KUKA KRL program: EPS_2_25252_SD2A_A_20250910061719.src

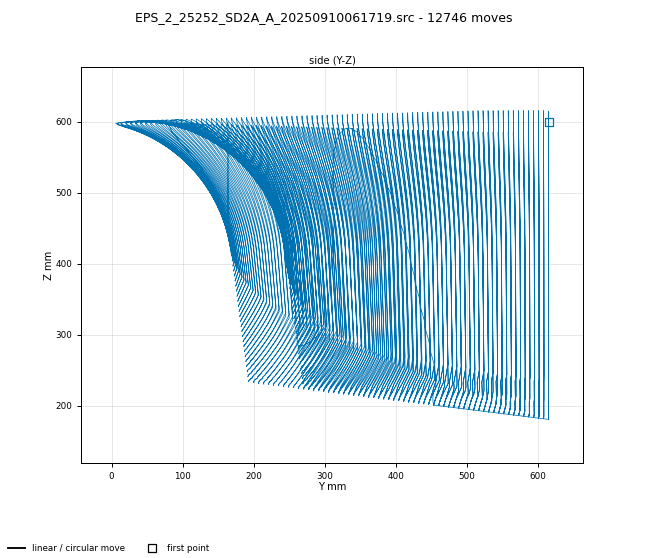
[picture p0: tool path of EPS_2_25252_SD2A_A_20250910061719.src, 12746 of 12748 moves have a stored position in this frame; points joined in program order, loops and branches not executed]
&ACCESS RVP
&REL 4
&COMMENT QRS 19112012
&PARAM EDITMASK = *
DEF PART()
EXT BAS (BAS_COMMAND :IN,REAL :IN )
INT I
BAS (#INITMOV,0 )

;KUKA QRS Post kuka4.cps  Date:22-06-2017 !

File_ID=2823

QRS_PRE_INIT()

;Init var - Until changes are made in qrs_pre_init
Outlet_Square_prg=0
Inlet_1_Square_prg=0
Inlet_2_Square_prg=0
Inlet_3_Square_prg=0
Inlet_4_Square_prg=0
Inlet_5_Square_prg=0

Outlet_1={X 0.000, Y 518.380, Z 433.000, B 0.000, E1 0.000 }
Inlet_1={X 0.000, Y 520.620, Z 403.000, B 0.000, E1 206.000 }
Outlet_1_type=366
Inlet_1_type=366
;QRS#1=Sidecore dimensions
;QRS#2=375-15" PVC SDR 35
;QRS#3=375-15" PVC SDR 35
;QRS#4=
;QRS#5=
;QRS#6=
;QRS#7=
;QRS#8=
;QRS#9=20Y PSX
;QRS#10=20Y PSX
;QRS#11=
;QRS#12=
;QRS#13=
;QRS#14=
;QRS#15=
;QRS#16=1220x127x914 3'
;QRS#17=EPS Height
;QRS#18=616
;QRS#19=*
;QRS#20= UPDATED VERSION 22-06-2017
;QRS#21=*
Outlet_Square=0250
Inlet_1_Square=0250
Inlet_2_Square=0
Inlet_3_Square=0
Inlet_4_Square=0
Inlet_5_Square=0
Mill_Square=1
Outlet_Square_Prg=252
Inlet_1_Square_prg=252

QRS_INIT()

$ADVANCE=5

; T1
PTP {E1 173.604,E2 173.604}
PTP {X 0,Y 615.505,A -85,B 0,C 180,E1 173.604,E2 173.604,E3 0,E4 0,E5 0,E6 0}
QRS_SPEED_INIT()
LIN {X 0,Y 615.505,Z 600,A -85,B 0,C 180,E1 173.604,E2 173.604,E3 0,E4 0,E5 0,E6 0} C_VEL
LIN {X 0,Y 615.505,Z 191.184,A -85,B 0,C 180,E1 173.604,E2 173.604} C_VEL
LIN {X 0,Y 615.505,Z 183.002,A -85,B 0,C 180,E1 173.604,E2 173.604} C_VEL
LIN {X 0,Y 615.487,Z 181.002,A -85,B 0,C 180,E1 173.418,E2 173.418} C_VEL
LIN {X 0,Y 615.475,Z 180.998,A -85,B 0,C 180,E1 170.801,E2 170.801} C_VEL
LIN {X 0,Y 615.481,Z 181.009,A -85,B 0,C 180,E1 168.139,E2 168.139} C_VEL
LIN {X 0,Y 615.486,Z 181,A -85,B 0,C 180,E1 165.451,E2 165.451} C_VEL
LIN {X 0,Y 615.47,Z 181.001,A -85,B 0,C 180,E1 162.729,E2 162.729} C_VEL
LIN {X 0,Y 615.488,Z 181.012,A -85,B 0,C 180,E1 159.967,E2 159.967} C_VEL
LIN {X 0,Y 615.49,Z 180.994,A -85,B 0,C 180,E1 157.156,E2 157.156} C_VEL
LIN {X 0,Y 615.489,Z 181.01,A -85,B 0,C 180,E1 154.284,E2 154.284} C_VEL
LIN {X 0,Y 615.487,Z 180.995,A -85,B 0,C 180,E1 151.342,E2 151.342} C_VEL
LIN {X 0,Y 615.474,Z 181,A -85,B 0,C 180,E1 148.915,E2 148.915} C_VEL
LIN {X 0,Y 615.485,Z 181.009,A -85,B 0,C 180,E1 146.465,E2 146.465} C_VEL
LIN {X 0,Y 615.482,Z 180.997,A -85,B 0,C 180,E1 143.575,E2 143.575} C_VEL
LIN {X 0,Y 615.474,Z 181.002,A -85,B 0,C 180,E1 140.939,E2 140.939} C_VEL
LIN {X 0,Y 615.488,Z 181.011,A -85,B 0,C 180,E1 138.526,E2 138.526} C_VEL
LIN {X 0,Y 615.477,Z 181,A -85,B 0,C 180,E1 135.85,E2 135.85} C_VEL
LIN {X 0,Y 615.477,Z 181.002,A -85,B 0,C 180,E1 133.047,E2 133.047} C_VEL
LIN {X 0,Y 615.491,Z 181.013,A -85,B 0,C 180,E1 130.606,E2 130.606} C_VEL
LIN {X 0,Y 615.477,Z 181.001,A -85,B 0,C 180,E1 128.011,E2 128.011} C_VEL
LIN {X 0,Y 615.497,Z 180.993,A -85,B 0,C 180,E1 125.615,E2 125.615} C_VEL
LIN {X 0,Y 615.48,Z 181.001,A -85,B 0,C 180,E1 123.236,E2 123.236} C_VEL
LIN {X 0,Y 615.486,Z 181.008,A -85,B 0,C 180,E1 120.92,E2 120.92} C_VEL
LIN {X 0,Y 615.476,Z 181.007,A -85,B 0,C 180,E1 118.449,E2 118.449} C_VEL
LIN {X 0,Y 615.489,Z 180.996,A -85,B 0,C 180,E1 115.569,E2 115.569} C_VEL
LIN {X 0,Y 615.487,Z 181.015,A -85,B 0,C 180,E1 112.844,E2 112.844} C_VEL
LIN {X 0,Y 615.48,Z 180.997,A -85,B 0,C 180,E1 110.033,E2 110.033} C_VEL
LIN {X 0,Y 615.484,Z 181.005,A -85,B 0,C 180,E1 107.271,E2 107.271} C_VEL
LIN {X 0,Y 615.472,Z 181.005,A -85,B 0,C 180,E1 104.549,E2 104.549} C_VEL
LIN {X 0,Y 615.486,Z 180.996,A -85,B 0,C 180,E1 101.861,E2 101.861} C_VEL
LIN {X 0,Y 615.489,Z 181.01,A -85,B 0,C 180,E1 99.199,E2 99.199} C_VEL
LIN {X 0,Y 615.468,Z 181.003,A -85,B 0,C 180,E1 96.557,E2 96.557} C_VEL
LIN {X 0,Y 615.487,Z 180.996,A -85,B 0,C 180,E1 93.929,E2 93.929} C_VEL
LIN {X 0,Y 615.489,Z 181.011,A -85,B 0,C 180,E1 91.309,E2 91.309} C_VEL
LIN {X 0,Y 615.465,Z 181.004,A -85,B 0,C 180,E1 88.692,E2 88.692} C_VEL
LIN {X 0,Y 615.48,Z 181.04,A -85,B 0,C 180,E1 88.242,E2 88.242} C_VEL
LIN {X 0,Y 615.493,Z 205.876,A -85,B 0,C 180,E1 85.969,E2 85.969} C_VEL
LIN {X 0,Y 615.49,Z 411.015,A -85,B 0,C 180,E1 83.444,E2 83.444} C_VEL
LIN {X 0,Y 615.494,Z 426.259,A -85,B 0,C 180,E1 83.141,E2 83.141} C_VEL
LIN {X 0,Y 615.491,Z 442.192,A -85,B 0,C 180,E1 82.702,E2 82.702} C_VEL
LIN {X 0,Y 615.493,Z 458.161,A -85,B 0,C 180,E1 82.125,E2 82.125} C_VEL
LIN {X 0,Y 615.492,Z 472.639,A -85,B 0,C 180,E1 81.464,E2 81.464} C_VEL
LIN {X 0,Y 615.498,Z 487.682,A -85,B 0,C 180,E1 80.636,E2 80.636} C_VEL
LIN {X 0,Y 615.495,Z 501.587,A -85,B 0,C 180,E1 79.723,E2 79.723} C_VEL
LIN {X 0,Y 615.496,Z 513.498,A -85,B 0,C 180,E1 78.807,E2 78.807} C_VEL
LIN {X 0,Y 615.493,Z 526.453,A -85,B 0,C 180,E1 77.638,E2 77.638} C_VEL
LIN {X 0,Y 615.498,Z 537.483,A -85,B 0,C 180,E1 76.463,E2 76.463} C_VEL
LIN {X 0,Y 615.491,Z 547.006,A -85,B 0,C 180,E1 75.282,E2 75.282} C_VEL
LIN {X 0,Y 615.492,Z 555.274,A -85,B 0,C 180,E1 74.095,E2 74.095} C_VEL
LIN {X 0,Y 615.49,Z 563.212,A -85,B 0,C 180,E1 72.73,E2 72.73} C_VEL
LIN {X 0,Y 615.491,Z 569.836,A -85,B 0,C 180,E1 71.355,E2 71.355} C_VEL
LIN {X 0,Y 615.491,Z 575.27,A -85,B 0,C 180,E1 69.968,E2 69.968} C_VEL
LIN {X 0,Y 615.497,Z 579.442,A -85,B 0,C 180,E1 68.569,E2 68.569} C_VEL
LIN {X 0,Y 615.485,Z 582.529,A -85,B 0,C 180,E1 67.156,E2 67.156} C_VEL
LIN {X 0,Y 615.486,Z 584.519,A -85,B 0,C 180,E1 65.728,E2 65.728} C_VEL
LIN {X 0,Y 615.5,Z 585.313,A -85,B 0,C 180,E1 64.285,E2 64.285} C_VEL
LIN {X 0,Y 615.485,Z 584.997,A -85,B 0,C 180,E1 62.823,E2 62.823} C_VEL
LIN {X 0,Y 615.485,Z 583.512,A -85,B 0,C 180,E1 61.343,E2 61.343} C_VEL
LIN {X 0,Y 615.486,Z 580.675,A -85,B 0,C 180,E1 59.84,E2 59.84} C_VEL
LIN {X 0,Y 615.495,Z 576.462,A -85,B 0,C 180,E1 58.316,E2 58.316} C_VEL
LIN {X 0,Y 615.488,Z 570.734,A -85,B 0,C 180,E1 56.765,E2 56.765} C_VEL
LIN {X 0,Y 615.49,Z 565.578,A -85,B 0,C 180,E1 55.64,E2 55.64} C_VEL
LIN {X 0,Y 615.499,Z 558.745,A -85,B 0,C 180,E1 54.386,E2 54.386} C_VEL
LIN {X 0,Y 615.492,Z 550.22,A -85,B 0,C 180,E1 53.063,E2 53.063} C_VEL
LIN {X 0,Y 615.494,Z 539.889,A -85,B 0,C 180,E1 51.725,E2 51.725} C_VEL
LIN {X 0,Y 615.499,Z 527.977,A -85,B 0,C 180,E1 50.424,E2 50.424} C_VEL
LIN {X 0,Y 615.493,Z 515.499,A -85,B 0,C 180,E1 49.273,E2 49.273} C_VEL
LIN {X 0,Y 615.499,Z 503.131,A -85,B 0,C 180,E1 48.3,E2 48.3} C_VEL
LIN {X 0,Y 615.495,Z 489.57,A -85,B 0,C 180,E1 47.388,E2 47.388} C_VEL
LIN {X 0,Y 615.493,Z 475.141,A -85,B 0,C 180,E1 46.569,E2 46.569} C_VEL
LIN {X 0,Y 615.493,Z 459.721,A -85,B 0,C 180,E1 45.852,E2 45.852} C_VEL
LIN {X 0,Y 615.496,Z 445.386,A -85,B 0,C 180,E1 45.315,E2 45.315} C_VEL
LIN {X 0,Y 615.49,Z 429.017,A -85,B 0,C 180,E1 44.834,E2 44.834} C_VEL
LIN {X 0,Y 615.494,Z 412.614,A -85,B 0,C 180,E1 44.49,E2 44.49} C_VEL
LIN {X 0,Y 615.451,Z 290.429,A -85,B 0,C 180,E1 42.979,E2 42.979} C_VEL
LIN {X 0,Y 615.445,Z 205.76,A -85,B 0,C 180,E1 41.928,E2 41.928} C_VEL
LIN {X 0,Y 615.419,Z 181.064,A -85,B 0,C 180,E1 39.668,E2 39.668} C_VEL
LIN {X 0,Y 615.463,Z 181.013,A -85,B 0,C 180,E1 36.935,E2 36.935} C_VEL
LIN {X 0,Y 615.496,Z 181.01,A -85,B 0,C 180,E1 34.703,E2 34.703} C_VEL
LIN {X 0,Y 615.426,Z 181.01,A -85,B 0,C 180,E1 31.689,E2 31.689} C_VEL
LIN {X 0,Y 615.444,Z 181.01,A -85,B 0,C 180,E1 29.408,E2 29.408} C_VEL
LIN {X 0,Y 615.462,Z 181.005,A -85,B 0,C 180,E1 26.445,E2 26.445} C_VEL
LIN {X 0,Y 615.437,Z 181.007,A -85,B 0,C 180,E1 24,E2 24} C_VEL
LIN {X 0,Y 615.442,Z 181.006,A -85,B 0,C 180,E1 22.138,E2 22.138} C_VEL
LIN {X 0,Y 615.439,Z 181.007,A -85,B 0,C 180,E1 20.034,E2 20.034} C_VEL
LIN {X 0,Y 615.491,Z 181.013,A -85,B 0,C 180,E1 17.27,E2 17.27} C_VEL
LIN {X 0,Y 615.468,Z 181.001,A -85,B 0,C 180,E1 14.549,E2 14.549} C_VEL
LIN {X 0,Y 615.465,Z 181.001,A -85,B 0,C 180,E1 12.531,E2 12.531} C_VEL
LIN {X 0,Y 615.46,Z 181.008,A -85,B 0,C 180,E1 9.863,E2 9.863} C_VEL
LIN {X 0,Y 615.493,Z 181.005,A -85,B 0,C 180,E1 7.216,E2 7.216} C_VEL
LIN {X 0,Y 615.462,Z 181.001,A -85,B 0,C 180,E1 4.585,E2 4.585} C_VEL
LIN {X 0,Y 615.47,Z 181.008,A -85,B 0,C 180,E1 1.963,E2 1.963} C_VEL
LIN {X 0,Y 615.489,Z 181.003,A -85,B 0,C 180,E1 -0.654,E2 -0.654} C_VEL
LIN {X 0,Y 615.474,Z 180.999,A -85,B 0,C 180,E1 -3.273,E2 -3.273} C_VEL
LIN {X 0,Y 615.472,Z 181.01,A -85,B 0,C 180,E1 -5.899,E2 -5.899} C_VEL
LIN {X 0,Y 615.484,Z 181.002,A -85,B 0,C 180,E1 -8.537,E2 -8.537} C_VEL
LIN {X 0,Y 615.476,Z 180.998,A -85,B 0,C 180,E1 -11.193,E2 -11.193} C_VEL
LIN {X 0,Y 615.499,Z 181.012,A -85,B 0,C 180,E1 -13.941,E2 -13.941} C_VEL
LIN {X 0,Y 615.486,Z 180.998,A -85,B 0,C 180,E1 -16.587,E2 -16.587} C_VEL
LIN {X 0,Y 615.474,Z 181.004,A -85,B 0,C 180,E1 -19.338,E2 -19.338} C_VEL
LIN {X 0,Y 615.478,Z 181.005,A -85,B 0,C 180,E1 -22.137,E2 -22.137} C_VEL
LIN {X 0,Y 615.483,Z 180.998,A -85,B 0,C 180,E1 -24.992,E2 -24.992} C_VEL
LIN {X 0,Y 615.475,Z 181.007,A -85,B 0,C 180,E1 -27.916,E2 -27.916} C_VEL
LIN {X 0,Y 615.47,Z 181.002,A -85,B 0,C 180,E1 -30.161,E2 -30.161} C_VEL
LIN {X 0,Y 615.484,Z 180.996,A -85,B 0,C 180,E1 -32.458,E2 -32.458} C_VEL
LIN {X 0,Y 615.487,Z 180.999,A -85,B 0,C 180,E1 -34.815,E2 -34.815} C_VEL
LIN {X 0,Y 615.487,Z 181.011,A -85,B 0,C 180,E1 -37.242,E2 -37.242} C_VEL
LIN {X 0,Y 615.466,Z 181.001,A -85,B 0,C 180,E1 -40.088,E2 -40.088} C_VEL
LIN {X 0,Y 615.482,Z 180.997,A -85,B 0,C 180,E1 -42.353,E2 -42.353} C_VEL
LIN {X 0,Y 615.492,Z 181.011,A -85,B 0,C 180,E1 -45.068,E2 -45.068} C_VEL
LIN {X 0,Y 615.458,Z 181.006,A -85,B 0,C 180,E1 -47.645,E2 -47.645} C_VEL
LIN {X 0,Y 615.479,Z 180.998,A -85,B 0,C 180,E1 -50.25,E2 -50.25} C_VEL
LIN {X 0,Y 615.486,Z 181.011,A -85,B 0,C 180,E1 -53.063,E2 -53.063} C_VEL
LIN {X 0,Y 615.458,Z 181.009,A -85,B 0,C 180,E1 -55.303,E2 -55.303} C_VEL
LIN {X 0,Y 615.448,Z 181.005,A -85,B 0,C 180,E1 -57.675,E2 -57.675} C_VEL
LIN {X 0,Y 615.482,Z 181.001,A -85,B 0,C 180,E1 -60.206,E2 -60.206} C_VEL
LIN {X 0,Y 615.468,Z 181.011,A -85,B 0,C 180,E1 -62.958,E2 -62.958} C_VEL
LIN {X 0,Y 615.442,Z 181.191,A -85,B 0,C 180,E1 -63.6,E2 -63.6} C_VEL
LIN {X 0,Y 615.497,Z 213.169,A -85,B 0,C 180,E1 -66.218,E2 -66.218} C_VEL
LIN {X 0,Y 615.485,Z 235.018,A -85,B 0,C 180,E1 -67.974,E2 -67.974} C_VEL
LIN {X 0,Y 615.49,Z 442.459,A -85,B 0,C 180,E1 -70.533,E2 -70.533} C_VEL
LIN {X 0,Y 615.493,Z 459.015,A -85,B 0,C 180,E1 -70.879,E2 -70.879} C_VEL
LIN {X 0,Y 615.492,Z 473.946,A -85,B 0,C 180,E1 -71.311,E2 -71.311} C_VEL
LIN {X 0,Y 615.491,Z 489.356,A -85,B 0,C 180,E1 -71.881,E2 -71.881} C_VEL
LIN {X 0,Y 615.493,Z 504.014,A -85,B 0,C 180,E1 -72.559,E2 -72.559} C_VEL
LIN {X 0,Y 615.5,Z 517.843,A -85,B 0,C 180,E1 -73.329,E2 -73.329} C_VEL
LIN {X 0,Y 615.499,Z 532.043,A -85,B 0,C 180,E1 -74.266,E2 -74.266} C_VEL
LIN {X 0,Y 615.495,Z 545.097,A -85,B 0,C 180,E1 -75.282,E2 -75.282} C_VEL
LIN {X 0,Y 615.494,Z 556.218,A -85,B 0,C 180,E1 -76.295,E2 -76.295} C_VEL
LIN {X 0,Y 615.493,Z 567.294,A -85,B 0,C 180,E1 -77.47,E2 -77.47} C_VEL
LIN {X 0,Y 615.494,Z 576.769,A -85,B 0,C 180,E1 -78.641,E2 -78.641} C_VEL
LIN {X 0,Y 615.496,Z 585.966,A -85,B 0,C 180,E1 -79.972,E2 -79.972} C_VEL
LIN {X 0,Y 615.489,Z 594.503,A -85,B 0,C 180,E1 -81.464,E2 -81.464} C_VEL
LIN {X 0,Y 615.491,Z 601.983,A -85,B 0,C 180,E1 -83.102,E2 -83.102} C_VEL
LIN {X 0,Y 615.492,Z 607.742,A -85,B 0,C 180,E1 -84.759,E2 -84.759} C_VEL
LIN {X 0,Y 615.493,Z 611.077,A -85,B 0,C 180,E1 -86.072,E2 -86.072} C_VEL
LIN {X 0,Y 615.485,Z 613.504,A -85,B 0,C 180,E1 -87.382,E2 -87.382} C_VEL
LIN {X 0,Y 615.488,Z 614.87,A -85,B 0,C 180,E1 -88.692,E2 -88.692} C_VEL
LIN {X 0,Y 615.489,Z 615.39,A -85,B 0,C 180,E1 -90,E2 -90} C_VEL
LIN {X 0,Y 615.488,Z 614.87,A -85,B 0,C 180,E1 -91.309,E2 -91.309} C_VEL
LIN {X 0,Y 615.485,Z 613.504,A -85,B 0,C 180,E1 -92.618,E2 -92.618} C_VEL
LIN {X 0,Y 615.493,Z 611.076,A -85,B 0,C 180,E1 -93.929,E2 -93.929} C_VEL
LIN {X 0,Y 615.492,Z 607.741,A -85,B 0,C 180,E1 -95.241,E2 -95.241} C_VEL
LIN {X 0,Y 615.491,Z 601.982,A -85,B 0,C 180,E1 -96.898,E2 -96.898} C_VEL
LIN {X 0,Y 615.489,Z 594.501,A -85,B 0,C 180,E1 -98.537,E2 -98.537} C_VEL
LIN {X 0,Y 615.496,Z 585.964,A -85,B 0,C 180,E1 -100.028,E2 -100.028} C_VEL
LIN {X 0,Y 615.494,Z 576.766,A -85,B 0,C 180,E1 -101.36,E2 -101.36} C_VEL
LIN {X 0,Y 615.495,Z 567.29,A -85,B 0,C 180,E1 -102.53,E2 -102.53} C_VEL
LIN {X 0,Y 615.496,Z 556.213,A -85,B 0,C 180,E1 -103.706,E2 -103.706} C_VEL
LIN {X 0,Y 615.495,Z 544.115,A -85,B 0,C 180,E1 -104.802,E2 -104.802} C_VEL
LIN {X 0,Y 615.497,Z 529.708,A -85,B 0,C 180,E1 -105.905,E2 -105.905} C_VEL
LIN {X 0,Y 615.497,Z 515.015,A -85,B 0,C 180,E1 -106.842,E2 -106.842} C_VEL
LIN {X 0,Y 615.49,Z 500.511,A -85,B 0,C 180,E1 -107.613,E2 -107.613} C_VEL
LIN {X 0,Y 615.49,Z 485.248,A -85,B 0,C 180,E1 -108.282,E2 -108.282} C_VEL
LIN {X 0,Y 615.49,Z 469.995,A -85,B 0,C 180,E1 -108.819,E2 -108.819} C_VEL
LIN {X 0,Y 615.497,Z 453.521,A -85,B 0,C 180,E1 -109.251,E2 -109.251} C_VEL
LIN {X 0,Y 615.49,Z 437.931,A -85,B 0,C 180,E1 -109.533,E2 -109.533} C_VEL
LIN {X 0,Y 615.485,Z 235.013,A -85,B 0,C 180,E1 -112.026,E2 -112.026} C_VEL
LIN {X 0,Y 615.453,Z 201.612,A -85,B 0,C 180,E1 -114.723,E2 -114.723} C_VEL
LIN {X 0,Y 615.441,Z 181.006,A -85,B 0,C 180,E1 -116.423,E2 -116.423} C_VEL
LIN {X 0,Y 615.443,Z 181.008,A -85,B 0,C 180,E1 -118.66,E2 -118.66} C_VEL
LIN {X 0,Y 615.477,Z 181.011,A -85,B 0,C 180,E1 -121.085,E2 -121.085} C_VEL
LIN {X 0,Y 615.457,Z 181.003,A -85,B 0,C 180,E1 -124.024,E2 -124.024} C_VEL
LIN {X 0,Y 615.444,Z 181.006,A -85,B 0,C 180,E1 -126.427,E2 -126.427} C_VEL
LIN {X 0,Y 615.492,Z 181.012,A -85,B 0,C 180,E1 -129.063,E2 -129.063} C_VEL
LIN {X 0,Y 615.494,Z 181.001,A -85,B 0,C 180,E1 -131.473,E2 -131.473} C_VEL
LIN {X 0,Y 615.448,Z 181.004,A -85,B 0,C 180,E1 -134.153,E2 -134.153} C_VEL
LIN {X 0,Y 615.469,Z 181.011,A -85,B 0,C 180,E1 -136.754,E2 -136.754} C_VEL
LIN {X 0,Y 615.494,Z 181,A -85,B 0,C 180,E1 -139.394,E2 -139.394} C_VEL
LIN {X 0,Y 615.453,Z 181.003,A -85,B 0,C 180,E1 -141.992,E2 -141.992} C_VEL
LIN {X 0,Y 615.454,Z 181.008,A -85,B 0,C 180,E1 -144.382,E2 -144.382} C_VEL
LIN {X 0,Y 615.481,Z 181.014,A -85,B 0,C 180,E1 -146.764,E2 -146.764} C_VEL
LIN {X 0,Y 615.493,Z 181.004,A -85,B 0,C 180,E1 -149.081,E2 -149.081} C_VEL
LIN {X 0,Y 615.474,Z 180.999,A -85,B 0,C 180,E1 -151.551,E2 -151.551} C_VEL
LIN {X 0,Y 615.469,Z 181,A -85,B 0,C 180,E1 -153.555,E2 -153.555} C_VEL
LIN {X 0,Y 615.455,Z 181.004,A -85,B 0,C 180,E1 -155.997,E2 -155.997} C_VEL
LIN {X 0,Y 615.491,Z 181.012,A -85,B 0,C 180,E1 -158.568,E2 -158.568} C_VEL
LIN {X 0,Y 615.477,Z 180.998,A -85,B 0,C 180,E1 -161.396,E2 -161.396} C_VEL
LIN {X 0,Y 615.463,Z 181.007,A -85,B 0,C 180,E1 -164.094,E2 -164.094} C_VEL
LIN {X 0,Y 615.487,Z 181.005,A -85,B 0,C 180,E1 -166.799,E2 -166.799} C_VEL
LIN {X 0,Y 615.468,Z 180.999,A -85,B 0,C 180,E1 -169.473,E2 -169.473} C_VEL
LIN {X 0,Y 615.473,Z 181.009,A -85,B 0,C 180,E1 -172.124,E2 -172.124} C_VEL
LIN {X 0,Y 615.489,Z 181.002,A -85,B 0,C 180,E1 -174.759,E2 -174.759} C_VEL
LIN {X 0,Y 615.47,Z 180.999,A -85,B 0,C 180,E1 -177.382,E2 -177.382} C_VEL
LIN {X 0,Y 615.475,Z 181.009,A -85,B 0,C 180,E1 -180,E2 -180} C_VEL
LIN {X 0,Y 615.488,Z 181.003,A -85,B 0,C 180,E1 -182.618,E2 -182.618} C_VEL
LIN {X 0,Y 615.474,Z 180.998,A -85,B 0,C 180,E1 -185.241,E2 -185.241} C_VEL
LIN {X 0,Y 615.487,Z 181.002,A -85,B 0,C 180,E1 -186.582,E2 -186.582} C_VEL
LIN {X 0,Y 614.803,Z 181.145,A -85,B 0,C 180,E1 -187.128,E2 -187.128} C_VEL
LIN {X 0,Y 611.964,Z 181.571,A -85,B 0,C 180,E1 -188.014,E2 -188.014} C_VEL
LIN {X 0,Y 609.572,Z 181.876,A -85,B 0,C 180,E1 -188.727,E2 -188.727} C_VEL
LIN {X 0,Y 608.538,Z 181.991,A -85,B 0,C 180,E1 -189.276,E2 -189.276} C_VEL
LIN {X 0,Y 608.449,Z 182.002,A -85,B 0,C 180,E1 -189.463,E2 -189.463} C_VEL
LIN {X 0,Y 608.458,Z 182.009,A -85,B 0,C 180,E1 -192,E2 -192} C_VEL
LIN {X 0,Y 608.471,Z 181.999,A -85,B 0,C 180,E1 -194.721,E2 -194.721} C_VEL
LIN {X 0,Y 608.444,Z 182.003,A -85,B 0,C 180,E1 -197.477,E2 -197.477} C_VEL
LIN {X 0,Y 608.463,Z 182.003,A -85,B 0,C 180,E1 -200.274,E2 -200.274} C_VEL
LIN {X 0,Y 608.449,Z 182.001,A -85,B 0,C 180,E1 -203.124,E2 -203.124} C_VEL
LIN {X 0,Y 608.47,Z 182.006,A -85,B 0,C 180,E1 -205.722,E2 -205.722} C_VEL
LIN {X 0,Y 608.473,Z 181.998,A -85,B 0,C 180,E1 -208.621,E2 -208.621} C_VEL
LIN {X 0,Y 608.442,Z 182.005,A -85,B 0,C 180,E1 -211.318,E2 -211.318} C_VEL
LIN {X 0,Y 608.471,Z 182.008,A -85,B 0,C 180,E1 -213.735,E2 -213.735} C_VEL
LIN {X 0,Y 608.474,Z 182.001,A -85,B 0,C 180,E1 -216.09,E2 -216.09} C_VEL
LIN {X 0,Y 608.462,Z 181.998,A -85,B 0,C 180,E1 -218.588,E2 -218.588} C_VEL
LIN {X 0,Y 608.458,Z 182.006,A -85,B 0,C 180,E1 -221.342,E2 -221.342} C_VEL
LIN {X 0,Y 608.447,Z 182.001,A -85,B 0,C 180,E1 -224.263,E2 -224.263} C_VEL
LIN {X 0,Y 608.445,Z 182.004,A -85,B 0,C 180,E1 -227.04,E2 -227.04} C_VEL
LIN {X 0,Y 608.45,Z 182.006,A -85,B 0,C 180,E1 -229.697,E2 -229.697} C_VEL
LIN {X 0,Y 608.462,Z 181.999,A -85,B 0,C 180,E1 -232.254,E2 -232.254} C_VEL
LIN {X 0,Y 608.48,Z 182.002,A -85,B 0,C 180,E1 -235.09,E2 -235.09} C_VEL
LIN {X 0,Y 608.462,Z 182,A -85,B 0,C 180,E1 -237.906,E2 -237.906} C_VEL
LIN {X 0,Y 608.472,Z 181.997,A -85,B 0,C 180,E1 -240.221,E2 -240.221} C_VEL
LIN {X 0,Y 608.476,Z 182.001,A -85,B 0,C 180,E1 -242.793,E2 -242.793} C_VEL
LIN {X 0,Y 608.447,Z 182.007,A -85,B 0,C 180,E1 -245.429,E2 -245.429} C_VEL
LIN {X 0,Y 608.463,Z 181.999,A -85,B 0,C 180,E1 -248.308,E2 -248.308} C_VEL
LIN {X 0,Y 608.466,Z 182.005,A -85,B 0,C 180,E1 -251.285,E2 -251.285} C_VEL
LIN {X 0,Y 608.454,Z 182,A -85,B 0,C 180,E1 -253.906,E2 -253.906} C_VEL
LIN {X 0,Y 608.467,Z 182.002,A -85,B 0,C 180,E1 -256.644,E2 -256.644} C_VEL
LIN {X 0,Y 608.453,Z 182.004,A -85,B 0,C 180,E1 -259.35,E2 -259.35} C_VEL
LIN {X 0,Y 608.476,Z 181.997,A -85,B 0,C 180,E1 -262.033,E2 -262.033} C_VEL
LIN {X 0,Y 608.47,Z 182.006,A -85,B 0,C 180,E1 -264.698,E2 -264.698} C_VEL
LIN {X 0,Y 608.459,Z 182.002,A -85,B 0,C 180,E1 -267.352,E2 -267.352} C_VEL
LIN {X 0,Y 608.477,Z 181.998,A -85,B 0,C 180,E1 -270,E2 -270} C_VEL
LIN {X 0,Y 608.461,Z 182.016,A -85,B 0,C 180,E1 -271.551,E2 -271.551} C_VEL
LIN {X 0,Y 608.729,Z 188.319,A -85,B 0,C 180,E1 -272.15,E2 -272.15} C_VEL
LIN {X 0,Y 608.693,Z 205.803,A -85,B 0,C 180,E1 -273.765,E2 -273.765} C_VEL
LIN {X 0,Y 608.912,Z 211.078,A -85,B 0,C 180,E1 -273.846,E2 -273.846} C_VEL
LIN {X 0,Y 608.803,Z 412.294,A -85,B 0,C 180,E1 -276.353,E2 -276.353} C_VEL
LIN {X 0,Y 608.775,Z 429.342,A -85,B 0,C 180,E1 -276.712,E2 -276.712} C_VEL
LIN {X 0,Y 608.754,Z 444.809,A -85,B 0,C 180,E1 -277.17,E2 -277.17} C_VEL
LIN {X 0,Y 608.708,Z 459.277,A -85,B 0,C 180,E1 -277.713,E2 -277.713} C_VEL
LIN {X 0,Y 608.657,Z 475.298,A -85,B 0,C 180,E1 -278.466,E2 -278.466} C_VEL
LIN {X 0,Y 608.63,Z 489.854,A -85,B 0,C 180,E1 -279.303,E2 -279.303} C_VEL
LIN {X 0,Y 608.57,Z 503.407,A -85,B 0,C 180,E1 -280.227,E2 -280.227} C_VEL
LIN {X 0,Y 608.53,Z 517.029,A -85,B 0,C 180,E1 -281.322,E2 -281.322} C_VEL
LIN {X 0,Y 608.494,Z 529.517,A -85,B 0,C 180,E1 -282.507,E2 -282.507} C_VEL
LIN {X 0,Y 608.475,Z 540.244,A -85,B 0,C 180,E1 -283.696,E2 -283.696} C_VEL
LIN {X 0,Y 608.477,Z 550.702,A -85,B 0,C 180,E1 -285.062,E2 -285.062} C_VEL
LIN {X 0,Y 608.438,Z 559.99,A -85,B 0,C 180,E1 -286.52,E2 -286.52} C_VEL
LIN {X 0,Y 608.45,Z 566.873,A -85,B 0,C 180,E1 -287.823,E2 -287.823} C_VEL
LIN {X 0,Y 608.434,Z 573.003,A -85,B 0,C 180,E1 -289.22,E2 -289.22} C_VEL
LIN {X 0,Y 608.434,Z 578.015,A -85,B 0,C 180,E1 -290.671,E2 -290.671} C_VEL
LIN {X 0,Y 608.423,Z 580.81,A -85,B 0,C 180,E1 -291.693,E2 -291.693} C_VEL
LIN {X 0,Y 608.425,Z 583.632,A -85,B 0,C 180,E1 -293.124,E2 -293.124} C_VEL
LIN {X 0,Y 608.402,Z 585.372,A -85,B 0,C 180,E1 -294.573,E2 -294.573} C_VEL
LIN {X 0,Y 608.419,Z 586,A -85,B 0,C 180,E1 -296.036,E2 -296.036} C_VEL
LIN {X 0,Y 608.42,Z 585.371,A -85,B 0,C 180,E1 -297.519,E2 -297.519} C_VEL
LIN {X 0,Y 608.404,Z 583.537,A -85,B 0,C 180,E1 -299.023,E2 -299.023} C_VEL
LIN {X 0,Y 608.422,Z 580.419,A -85,B 0,C 180,E1 -300.547,E2 -300.547} C_VEL
LIN {X 0,Y 608.427,Z 577.099,A -85,B 0,C 180,E1 -301.706,E2 -301.706} C_VEL
LIN {X 0,Y 608.431,Z 571.346,A -85,B 0,C 180,E1 -303.275,E2 -303.275} C_VEL
LIN {X 0,Y 608.434,Z 564.827,A -85,B 0,C 180,E1 -304.687,E2 -304.687} C_VEL
LIN {X 0,Y 608.451,Z 556.844,A -85,B 0,C 180,E1 -306.091,E2 -306.091} C_VEL
LIN {X 0,Y 608.477,Z 547.824,A -85,B 0,C 180,E1 -307.421,E2 -307.421} C_VEL
LIN {X 0,Y 608.496,Z 536.759,A -85,B 0,C 180,E1 -308.797,E2 -308.797} C_VEL
LIN {X 0,Y 608.533,Z 524.523,A -85,B 0,C 180,E1 -310.079,E2 -310.079} C_VEL
LIN {X 0,Y 608.551,Z 512.324,A -85,B 0,C 180,E1 -311.168,E2 -311.168} C_VEL
LIN {X 0,Y 608.591,Z 499.367,A -85,B 0,C 180,E1 -312.159,E2 -312.159} C_VEL
LIN {X 0,Y 608.644,Z 484.171,A -85,B 0,C 180,E1 -313.135,E2 -313.135} C_VEL
LIN {X 0,Y 608.688,Z 468.85,A -85,B 0,C 180,E1 -313.944,E2 -313.944} C_VEL
LIN {X 0,Y 608.73,Z 453.448,A -85,B 0,C 180,E1 -314.608,E2 -314.608} C_VEL
LIN {X 0,Y 608.761,Z 436.634,A -85,B 0,C 180,E1 -315.177,E2 -315.177} C_VEL
LIN {X 0,Y 608.807,Z 420.377,A -85,B 0,C 180,E1 -315.584,E2 -315.584} C_VEL
LIN {X 0,Y 608.827,Z 403.651,A -85,B 0,C 180,E1 -315.863,E2 -315.863} C_VEL
LIN {X 0,Y 608.847,Z 207.061,A -85,B 0,C 180,E1 -318.296,E2 -318.296} C_VEL
LIN {X 0,Y 608.641,Z 205.738,A -85,B 0,C 180,E1 -318.333,E2 -318.333} C_VEL
LIN {X 0,Y 608.678,Z 183.809,A -85,B 0,C 180,E1 -320.362,E2 -320.362} C_VEL
LIN {X 0,Y 608.4,Z 182.01,A -85,B 0,C 180,E1 -320.555,E2 -320.555} C_VEL
LIN {X 0,Y 608.434,Z 182.01,A -85,B 0,C 180,E1 -323.084,E2 -323.084} C_VEL
LIN {X 0,Y 608.461,Z 182.004,A -85,B 0,C 180,E1 -325.53,E2 -325.53} C_VEL
LIN {X 0,Y 608.431,Z 182.004,A -85,B 0,C 180,E1 -327.904,E2 -327.904} C_VEL
LIN {X 0,Y 608.417,Z 182.005,A -85,B 0,C 180,E1 -330.218,E2 -330.218} C_VEL
LIN {X 0,Y 608.449,Z 182.007,A -85,B 0,C 180,E1 -332.796,E2 -332.796} C_VEL
LIN {X 0,Y 608.438,Z 182.005,A -85,B 0,C 180,E1 -335.428,E2 -335.428} C_VEL
LIN {X 0,Y 608.438,Z 182.004,A -85,B 0,C 180,E1 -338.307,E2 -338.307} C_VEL
LIN {X 0,Y 608.462,Z 182.002,A -85,B 0,C 180,E1 -341.284,E2 -341.284} C_VEL
LIN {X 0,Y 608.429,Z 182.003,A -85,B 0,C 180,E1 -343.905,E2 -343.905} C_VEL
LIN {X 0,Y 608.462,Z 182.009,A -85,B 0,C 180,E1 -346.644,E2 -346.644} C_VEL
LIN {X 0,Y 608.451,Z 182.001,A -85,B 0,C 180,E1 -349.35,E2 -349.35} C_VEL
LIN {X 0,Y 608.456,Z 182.003,A -85,B 0,C 180,E1 -352.033,E2 -352.033} C_VEL
LIN {X 0,Y 608.465,Z 182.005,A -85,B 0,C 180,E1 -354.698,E2 -354.698} C_VEL
LIN {X 0,Y 608.461,Z 181.999,A -85,B 0,C 180,E1 -357.352,E2 -357.352} C_VEL
LIN {X 0,Y 608.463,Z 182.004,A -85,B 0,C 180,E1 -360,E2 -360} C_VEL
LIN {X 0,Y 608.478,Z 182.001,A -85,B 0,C 180,E1 -362.648,E2 -362.648} C_VEL
LIN {X 0,Y 608.453,Z 182,A -85,B 0,C 180,E1 -365.302,E2 -365.302} C_VEL
LIN {X 0,Y 608.472,Z 182.006,A -85,B 0,C 180,E1 -367.967,E2 -367.967} C_VEL
LIN {X 0,Y 608.466,Z 181.998,A -85,B 0,C 180,E1 -370.959,E2 -370.959} C_VEL
LIN {X 0,Y 608.458,Z 182.001,A -85,B 0,C 180,E1 -373.356,E2 -373.356} C_VEL
LIN {X 0,Y 608.459,Z 182.006,A -85,B 0,C 180,E1 -376.094,E2 -376.094} C_VEL
LIN {X 0,Y 608.45,Z 182,A -85,B 0,C 180,E1 -378.87,E2 -378.87} C_VEL
LIN {X 0,Y 608.461,Z 182.009,A -85,B 0,C 180,E1 -381.692,E2 -381.692} C_VEL
LIN {X 0,Y 608.446,Z 182.001,A -85,B 0,C 180,E1 -384.571,E2 -384.571} C_VEL
LIN {X 0,Y 608.474,Z 182.001,A -85,B 0,C 180,E1 -387.208,E2 -387.208} C_VEL
LIN {X 0,Y 608.458,Z 182.003,A -85,B 0,C 180,E1 -389.972,E2 -389.972} C_VEL
LIN {X 0,Y 608.459,Z 181.999,A -85,B 0,C 180,E1 -392.523,E2 -392.523} C_VEL
LIN {X 0,Y 608.441,Z 182.01,A -85,B 0,C 180,E1 -395.278,E2 -395.278} C_VEL
LIN {X 0,Y 608.457,Z 182.003,A -85,B 0,C 180,E1 -397.747,E2 -397.747} C_VEL
LIN {X 0,Y 608.444,Z 182.001,A -85,B 0,C 180,E1 -400.329,E2 -400.329} C_VEL
LIN {X 0,Y 608.48,Z 182.005,A -85,B 0,C 180,E1 -403.311,E2 -403.311} C_VEL
LIN {X 0,Y 608.452,Z 182,A -85,B 0,C 180,E1 -406.13,E2 -406.13} C_VEL
LIN {X 0,Y 608.463,Z 182.005,A -85,B 0,C 180,E1 -408.825,E2 -408.825} C_VEL
LIN {X 0,Y 608.433,Z 182.006,A -85,B 0,C 180,E1 -411.41,E2 -411.41} C_VEL
LIN {X 0,Y 608.437,Z 182.002,A -85,B 0,C 180,E1 -413.955,E2 -413.955} C_VEL
LIN {X 0,Y 608.461,Z 182.001,A -85,B 0,C 180,E1 -416.33,E2 -416.33} C_VEL
LIN {X 0,Y 608.475,Z 182.007,A -85,B 0,C 180,E1 -418.728,E2 -418.728} C_VEL
LIN {X 0,Y 608.438,Z 182.004,A -85,B 0,C 180,E1 -421.386,E2 -421.386} C_VEL
LIN {X 0,Y 608.432,Z 182.019,A -85,B 0,C 180,E1 -423.341,E2 -423.341} C_VEL
LIN {X 0,Y 608.799,Z 186.159,A -85,B 0,C 180,E1 -423.705,E2 -423.705} C_VEL
LIN {X 0,Y 608.748,Z 219.284,A -85,B 0,C 180,E1 -426.438,E2 -426.438} C_VEL
LIN {X 0,Y 608.704,Z 235.018,A -85,B 0,C 180,E1 -427.716,E2 -427.716} C_VEL
LIN {X 0,Y 608.928,Z 247.383,A -85,B 0,C 180,E1 -427.881,E2 -427.881} C_VEL
LIN {X 0,Y 608.795,Z 440.971,A -85,B 0,C 180,E1 -430.288,E2 -430.288} C_VEL
LIN {X 0,Y 608.795,Z 457.191,A -85,B 0,C 180,E1 -430.617,E2 -430.617} C_VEL
LIN {X 0,Y 608.737,Z 472.657,A -85,B 0,C 180,E1 -431.053,E2 -431.053} C_VEL
LIN {X 0,Y 608.711,Z 487.377,A -85,B 0,C 180,E1 -431.59,E2 -431.59} C_VEL
LIN {X 0,Y 608.678,Z 502.27,A -85,B 0,C 180,E1 -432.27,E2 -432.27} C_VEL
LIN {X 0,Y 608.616,Z 517.846,A -85,B 0,C 180,E1 -433.135,E2 -433.135} C_VEL
LIN {X 0,Y 608.578,Z 532.052,A -85,B 0,C 180,E1 -434.082,E2 -434.082} C_VEL
LIN {X 0,Y 608.556,Z 545.132,A -85,B 0,C 180,E1 -435.111,E2 -435.111} C_VEL
LIN {X 0,Y 608.528,Z 557.01,A -85,B 0,C 180,E1 -436.204,E2 -436.204} C_VEL
LIN {X 0,Y 608.49,Z 568.915,A -85,B 0,C 180,E1 -437.493,E2 -437.493} C_VEL
LIN {X 0,Y 608.486,Z 578.209,A -85,B 0,C 180,E1 -438.677,E2 -438.677} C_VEL
LIN {X 0,Y 608.471,Z 587.26,A -85,B 0,C 180,E1 -440.023,E2 -440.023} C_VEL
LIN {X 0,Y 608.444,Z 594.859,A -85,B 0,C 180,E1 -441.364,E2 -441.364} C_VEL
LIN {X 0,Y 608.437,Z 602.47,A -85,B 0,C 180,E1 -443.034,E2 -443.034} C_VEL
LIN {X 0,Y 608.435,Z 608.246,A -85,B 0,C 180,E1 -444.698,E2 -444.698} C_VEL
LIN {X 0,Y 608.43,Z 611.633,A -85,B 0,C 180,E1 -446.026,E2 -446.026} C_VEL
LIN {X 0,Y 608.412,Z 614.086,A -85,B 0,C 180,E1 -447.352,E2 -447.352} C_VEL
LIN {X 0,Y 608.441,Z 615.477,A -85,B 0,C 180,E1 -448.676,E2 -448.676} C_VEL
LIN {X 0,Y 608.429,Z 616,A -85,B 0,C 180,E1 -450,E2 -450} C_VEL
LIN {X 0,Y 608.441,Z 615.477,A -85,B 0,C 180,E1 -451.324,E2 -451.324} C_VEL
LIN {X 0,Y 608.412,Z 614.085,A -85,B 0,C 180,E1 -452.648,E2 -452.648} C_VEL
LIN {X 0,Y 608.43,Z 611.632,A -85,B 0,C 180,E1 -453.974,E2 -453.974} C_VEL
LIN {X 0,Y 608.435,Z 608.245,A -85,B 0,C 180,E1 -455.302,E2 -455.302} C_VEL
LIN {X 0,Y 608.437,Z 602.468,A -85,B 0,C 180,E1 -456.966,E2 -456.966} C_VEL
LIN {X 0,Y 608.444,Z 594.857,A -85,B 0,C 180,E1 -458.636,E2 -458.636} C_VEL
LIN {X 0,Y 608.461,Z 586.245,A -85,B 0,C 180,E1 -460.145,E2 -460.145} C_VEL
LIN {X 0,Y 608.467,Z 576.967,A -85,B 0,C 180,E1 -461.493,E2 -461.493} C_VEL
LIN {X 0,Y 608.49,Z 567.421,A -85,B 0,C 180,E1 -462.677,E2 -462.677} C_VEL
LIN {X 0,Y 608.524,Z 555.953,A -85,B 0,C 180,E1 -463.897,E2 -463.897} C_VEL
LIN {X 0,Y 608.553,Z 544.143,A -85,B 0,C 180,E1 -464.975,E2 -464.975} C_VEL
LIN {X 0,Y 608.607,Z 529.71,A -85,B 0,C 180,E1 -466.09,E2 -466.09} C_VEL
LIN {X 0,Y 608.623,Z 515.018,A -85,B 0,C 180,E1 -467.038,E2 -467.038} C_VEL
LIN {X 0,Y 608.66,Z 500.514,A -85,B 0,C 180,E1 -467.817,E2 -467.817} C_VEL
LIN {X 0,Y 608.718,Z 485.25,A -85,B 0,C 180,E1 -468.493,E2 -468.493} C_VEL
LIN {X 0,Y 608.748,Z 469.241,A -85,B 0,C 180,E1 -469.057,E2 -469.057} C_VEL
LIN {X 0,Y 608.786,Z 452.607,A -85,B 0,C 180,E1 -469.494,E2 -469.494} C_VEL
LIN {X 0,Y 608.806,Z 436.425,A -85,B 0,C 180,E1 -469.778,E2 -469.778} C_VEL
LIN {X 0,Y 608.911,Z 236.618,A -85,B 0,C 180,E1 -472.254,E2 -472.254} C_VEL
LIN {X 0,Y 608.72,Z 234.737,A -85,B 0,C 180,E1 -472.306,E2 -472.306} C_VEL
LIN {X 0,Y 608.774,Z 201.612,A -85,B 0,C 180,E1 -475.012,E2 -475.012} C_VEL
LIN {X 0,Y 608.81,Z 183.946,A -85,B 0,C 180,E1 -476.48,E2 -476.48} C_VEL
LIN {X 0,Y 608.416,Z 182.008,A -85,B 0,C 180,E1 -476.683,E2 -476.683} C_VEL
LIN {X 0,Y 608.466,Z 182.001,A -85,B 0,C 180,E1 -479.779,E2 -479.779} C_VEL
LIN {X 0,Y 608.425,Z 182.004,A -85,B 0,C 180,E1 -482.517,E2 -482.517} C_VEL
LIN {X 0,Y 608.429,Z 182.009,A -85,B 0,C 180,E1 -484.903,E2 -484.903} C_VEL
LIN {X 0,Y 608.454,Z 182.002,A -85,B 0,C 180,E1 -487.747,E2 -487.747} C_VEL
LIN {X 0,Y 608.429,Z 182.003,A -85,B 0,C 180,E1 -490.327,E2 -490.327} C_VEL
LIN {X 0,Y 608.447,Z 182.01,A -85,B 0,C 180,E1 -492.96,E2 -492.96} C_VEL
LIN {X 0,Y 608.434,Z 182.003,A -85,B 0,C 180,E1 -495.738,E2 -495.738} C_VEL
LIN {X 0,Y 608.438,Z 182.002,A -85,B 0,C 180,E1 -497.937,E2 -497.937} C_VEL
LIN {X 0,Y 608.44,Z 182.008,A -85,B 0,C 180,E1 -500.705,E2 -500.705} C_VEL
LIN {X 0,Y 608.464,Z 182.005,A -85,B 0,C 180,E1 -503.086,E2 -503.086} C_VEL
LIN {X 0,Y 608.465,Z 182,A -85,B 0,C 180,E1 -505.531,E2 -505.531} C_VEL
LIN {X 0,Y 608.447,Z 182,A -85,B 0,C 180,E1 -507.905,E2 -507.905} C_VEL
LIN {X 0,Y 608.44,Z 182.004,A -85,B 0,C 180,E1 -510.219,E2 -510.219} C_VEL
LIN {X 0,Y 608.481,Z 182.006,A -85,B 0,C 180,E1 -512.791,E2 -512.791} C_VEL
LIN {X 0,Y 608.443,Z 182.002,A -85,B 0,C 180,E1 -515.429,E2 -515.429} C_VEL
LIN {X 0,Y 608.46,Z 182.004,A -85,B 0,C 180,E1 -518.308,E2 -518.308} C_VEL
LIN {X 0,Y 608.465,Z 181.999,A -85,B 0,C 180,E1 -521.284,E2 -521.284} C_VEL
LIN {X 0,Y 608.44,Z 182.003,A -85,B 0,C 180,E1 -523.906,E2 -523.906} C_VEL
LIN {X 0,Y 608.46,Z 182.007,A -85,B 0,C 180,E1 -526.644,E2 -526.644} C_VEL
LIN {X 0,Y 608.453,Z 182,A -85,B 0,C 180,E1 -529.35,E2 -529.35} C_VEL
LIN {X 0,Y 608.465,Z 182.003,A -85,B 0,C 180,E1 -532.033,E2 -532.033} C_VEL
LIN {X 0,Y 608.467,Z 182.003,A -85,B 0,C 180,E1 -534.698,E2 -534.698} C_VEL
LIN {X 0,Y 608.463,Z 181.998,A -85,B 0,C 180,E1 -537.352,E2 -537.352} C_VEL
LIN {X 0,Y 608.467,Z 182.004,A -85,B 0,C 180,E1 -540,E2 -540} C_VEL
LIN {X 0,Y 608.478,Z 182,A -85,B 0,C 180,E1 -542.648,E2 -542.648} C_VEL
LIN {X 0,Y 608.453,Z 181.999,A -85,B 0,C 180,E1 -545.302,E2 -545.302} C_VEL
LIN {X 0,Y 608.47,Z 182.005,A -85,B 0,C 180,E1 -547.967,E2 -547.967} C_VEL
LIN {X 0,Y 608.449,Z 182.002,A -85,B 0,C 180,E1 -549.463,E2 -549.463} C_VEL
LIN {X 0,Y 607.771,Z 182.094,A -85,B 0,C 180,E1 -550.015,E2 -550.015} C_VEL
LIN {X 0,Y 604.919,Z 182.452,A -85,B 0,C 180,E1 -550.912,E2 -550.912} C_VEL
LIN {X 0,Y 602.519,Z 182.751,A -85,B 0,C 180,E1 -551.634,E2 -551.634} C_VEL
LIN {X 0,Y 601.489,Z 182.875,A -85,B 0,C 180,E1 -552.191,E2 -552.191} C_VEL
LIN {X 0,Y 601.405,Z 182.883,A -85,B 0,C 180,E1 -552.379,E2 -552.379} C_VEL
LIN {X 0,Y 601.425,Z 182.876,A -85,B 0,C 180,E1 -554.897,E2 -554.897} C_VEL
LIN {X 0,Y 601.427,Z 182.875,A -85,B 0,C 180,E1 -556.986,E2 -556.986} C_VEL
LIN {X 0,Y 601.401,Z 182.886,A -85,B 0,C 180,E1 -559.81,E2 -559.81} C_VEL
LIN {X 0,Y 601.412,Z 182.878,A -85,B 0,C 180,E1 -562.606,E2 -562.606} C_VEL
LIN {X 0,Y 601.397,Z 182.878,A -85,B 0,C 180,E1 -564.879,E2 -564.879} C_VEL
LIN {X 0,Y 601.418,Z 182.886,A -85,B 0,C 180,E1 -567.867,E2 -567.867} C_VEL
LIN {X 0,Y 601.446,Z 182.876,A -85,B 0,C 180,E1 -570.163,E2 -570.163} C_VEL
LIN {X 0,Y 601.42,Z 182.875,A -85,B 0,C 180,E1 -572.716,E2 -572.716} C_VEL
LIN {X 0,Y 601.41,Z 182.879,A -85,B 0,C 180,E1 -575.115,E2 -575.115} C_VEL
LIN {X 0,Y 601.43,Z 182.881,A -85,B 0,C 180,E1 -577.419,E2 -577.419} C_VEL
LIN {X 0,Y 601.399,Z 182.883,A -85,B 0,C 180,E1 -579.996,E2 -579.996} C_VEL
LIN {X 0,Y 601.408,Z 182.877,A -85,B 0,C 180,E1 -582.67,E2 -582.67} C_VEL
LIN {X 0,Y 601.424,Z 182.886,A -85,B 0,C 180,E1 -585.482,E2 -585.482} C_VEL
LIN {X 0,Y 601.421,Z 182.875,A -85,B 0,C 180,E1 -588.407,E2 -588.407} C_VEL
LIN {X 0,Y 601.427,Z 182.884,A -85,B 0,C 180,E1 -591.529,E2 -591.529} C_VEL
LIN {X 0,Y 601.389,Z 182.88,A -85,B 0,C 180,E1 -594.246,E2 -594.246} C_VEL
LIN {X 0,Y 601.425,Z 182.877,A -85,B 0,C 180,E1 -596.687,E2 -596.687} C_VEL
LIN {X 0,Y 601.419,Z 182.882,A -85,B 0,C 180,E1 -599.058,E2 -599.058} C_VEL
LIN {X 0,Y 601.43,Z 182.883,A -85,B 0,C 180,E1 -601.373,E2 -601.373} C_VEL
LIN {X 0,Y 601.418,Z 182.876,A -85,B 0,C 180,E1 -604.131,E2 -604.131} C_VEL
LIN {X 0,Y 601.42,Z 182.878,A -85,B 0,C 180,E1 -606.59,E2 -606.59} C_VEL
LIN {X 0,Y 601.425,Z 182.879,A -85,B 0,C 180,E1 -609.478,E2 -609.478} C_VEL
LIN {X 0,Y 601.396,Z 182.879,A -85,B 0,C 180,E1 -612.312,E2 -612.312} C_VEL
LIN {X 0,Y 601.424,Z 182.884,A -85,B 0,C 180,E1 -615.103,E2 -615.103} C_VEL
LIN {X 0,Y 601.414,Z 182.877,A -85,B 0,C 180,E1 -617.857,E2 -617.857} C_VEL
LIN {X 0,Y 601.421,Z 182.881,A -85,B 0,C 180,E1 -620.584,E2 -620.584} C_VEL
LIN {X 0,Y 601.401,Z 182.882,A -85,B 0,C 180,E1 -623.289,E2 -623.289} C_VEL
LIN {X 0,Y 601.406,Z 182.878,A -85,B 0,C 180,E1 -625.979,E2 -625.979} C_VEL
LIN {X 0,Y 601.427,Z 182.884,A -85,B 0,C 180,E1 -628.661,E2 -628.661} C_VEL
LIN {X 0,Y 601.438,Z 182.998,A -85,B 0,C 180,E1 -631.339,E2 -631.339} C_VEL
LIN {X 0,Y 601.988,Z 186.27,A -85,B 0,C 180,E1 -631.672,E2 -631.672} C_VEL
LIN {X 0,Y 601.887,Z 205.739,A -85,B 0,C 180,E1 -633.493,E2 -633.493} C_VEL
LIN {X 0,Y 602.354,Z 209.71,A -85,B 0,C 180,E1 -633.574,E2 -633.574} C_VEL
LIN {X 0,Y 602.117,Z 411.91,A -85,B 0,C 180,E1 -636.119,E2 -636.119} C_VEL
LIN {X 0,Y 602.076,Z 428.185,A -85,B 0,C 180,E1 -636.46,E2 -636.46} C_VEL
LIN {X 0,Y 602.013,Z 444.12,A -85,B 0,C 180,E1 -636.927,E2 -636.927} C_VEL
LIN {X 0,Y 601.932,Z 458.443,A -85,B 0,C 180,E1 -637.463,E2 -637.463} C_VEL
LIN {X 0,Y 601.858,Z 474.575,A -85,B 0,C 180,E1 -638.224,E2 -638.224} C_VEL
LIN {X 0,Y 601.755,Z 489.296,A -85,B 0,C 180,E1 -639.071,E2 -639.071} C_VEL
LIN {X 0,Y 601.669,Z 502.94,A -85,B 0,C 180,E1 -640.006,E2 -640.006} C_VEL
LIN {X 0,Y 601.577,Z 516.344,A -85,B 0,C 180,E1 -641.087,E2 -641.087} C_VEL
LIN {X 0,Y 601.545,Z 527.548,A -85,B 0,C 180,E1 -642.139,E2 -642.139} C_VEL
LIN {X 0,Y 601.484,Z 538.5,A -85,B 0,C 180,E1 -643.342,E2 -643.342} C_VEL
LIN {X 0,Y 601.436,Z 547.944,A -85,B 0,C 180,E1 -644.55,E2 -644.55} C_VEL
LIN {X 0,Y 601.41,Z 557.197,A -85,B 0,C 180,E1 -645.939,E2 -645.939} C_VEL
LIN {X 0,Y 601.394,Z 565.01,A -85,B 0,C 180,E1 -647.337,E2 -647.337} C_VEL
LIN {X 0,Y 601.376,Z 571.678,A -85,B 0,C 180,E1 -648.808,E2 -648.808} C_VEL
LIN {X 0,Y 601.332,Z 576.63,A -85,B 0,C 180,E1 -650.168,E2 -650.168} C_VEL
LIN {X 0,Y 601.322,Z 579.764,A -85,B 0,C 180,E1 -651.242,E2 -651.242} C_VEL
LIN {X 0,Y 601.318,Z 582.968,A -85,B 0,C 180,E1 -652.686,E2 -652.686} C_VEL
LIN {X 0,Y 601.307,Z 585.156,A -85,B 0,C 180,E1 -654.265,E2 -654.265} C_VEL
LIN {X 0,Y 601.334,Z 585.961,A -85,B 0,C 180,E1 -655.852,E2 -655.852} C_VEL
LIN {X 0,Y 601.344,Z 585.502,A -85,B 0,C 180,E1 -657.35,E2 -657.35} C_VEL
LIN {X 0,Y 601.329,Z 584.011,A -85,B 0,C 180,E1 -658.77,E2 -658.77} C_VEL
LIN {X 0,Y 601.337,Z 581.414,A -85,B 0,C 180,E1 -660.168,E2 -660.168} C_VEL
LIN {X 0,Y 601.342,Z 577.237,A -85,B 0,C 180,E1 -661.73,E2 -661.73} C_VEL
LIN {X 0,Y 601.365,Z 571.533,A -85,B 0,C 180,E1 -663.317,E2 -663.317} C_VEL
LIN {X 0,Y 601.368,Z 565.124,A -85,B 0,C 180,E1 -664.73,E2 -664.73} C_VEL
LIN {X 0,Y 601.382,Z 556.562,A -85,B 0,C 180,E1 -666.258,E2 -666.258} C_VEL
LIN {X 0,Y 601.442,Z 547.298,A -85,B 0,C 180,E1 -667.629,E2 -667.629} C_VEL
LIN {X 0,Y 601.485,Z 536.809,A -85,B 0,C 180,E1 -668.943,E2 -668.943} C_VEL
LIN {X 0,Y 601.534,Z 525.039,A -85,B 0,C 180,E1 -670.196,E2 -670.196} C_VEL
LIN {X 0,Y 601.6,Z 512.87,A -85,B 0,C 180,E1 -671.302,E2 -671.302} C_VEL
LIN {X 0,Y 601.703,Z 500.062,A -85,B 0,C 180,E1 -672.299,E2 -672.299} C_VEL
LIN {X 0,Y 601.768,Z 486.22,A -85,B 0,C 180,E1 -673.209,E2 -673.209} C_VEL
LIN {X 0,Y 601.859,Z 471.391,A -85,B 0,C 180,E1 -674.027,E2 -674.027} C_VEL
LIN {X 0,Y 601.939,Z 455.297,A -85,B 0,C 180,E1 -674.753,E2 -674.753} C_VEL
LIN {X 0,Y 602.029,Z 438.941,A -85,B 0,C 180,E1 -675.332,E2 -675.332} C_VEL
LIN {X 0,Y 602.094,Z 422.308,A -85,B 0,C 180,E1 -675.771,E2 -675.771} C_VEL
LIN {X 0,Y 602.129,Z 404.901,A -85,B 0,C 180,E1 -676.075,E2 -676.075} C_VEL
LIN {X 0,Y 602.303,Z 208.281,A -85,B 0,C 180,E1 -678.536,E2 -678.536} C_VEL
LIN {X 0,Y 601.84,Z 205.816,A -85,B 0,C 180,E1 -678.591,E2 -678.591} C_VEL
LIN {X 0,Y 601.925,Z 186.409,A -85,B 0,C 180,E1 -680.407,E2 -680.407} C_VEL
LIN {X 0,Y 601.362,Z 182.89,A -85,B 0,C 180,E1 -680.784,E2 -680.784} C_VEL
LIN {X 0,Y 601.38,Z 182.885,A -85,B 0,C 180,E1 -683.741,E2 -683.741} C_VEL
LIN {X 0,Y 601.396,Z 182.88,A -85,B 0,C 180,E1 -686.068,E2 -686.068} C_VEL
LIN {X 0,Y 601.402,Z 182.881,A -85,B 0,C 180,E1 -688.547,E2 -688.547} C_VEL
LIN {X 0,Y 601.424,Z 182.881,A -85,B 0,C 180,E1 -691.373,E2 -691.373} C_VEL
LIN {X 0,Y 601.382,Z 182.883,A -85,B 0,C 180,E1 -693.635,E2 -693.635} C_VEL
LIN {X 0,Y 601.42,Z 182.876,A -85,B 0,C 180,E1 -695.858,E2 -695.858} C_VEL
LIN {X 0,Y 601.393,Z 182.888,A -85,B 0,C 180,E1 -698.76,E2 -698.76} C_VEL
LIN {X 0,Y 601.384,Z 182.881,A -85,B 0,C 180,E1 -701.607,E2 -701.607} C_VEL
LIN {X 0,Y 601.413,Z 182.877,A -85,B 0,C 180,E1 -703.712,E2 -703.712} C_VEL
LIN {X 0,Y 601.404,Z 182.885,A -85,B 0,C 180,E1 -706.484,E2 -706.484} C_VEL
LIN {X 0,Y 601.409,Z 182.879,A -85,B 0,C 180,E1 -709.224,E2 -709.224} C_VEL
LIN {X 0,Y 601.421,Z 182.878,A -85,B 0,C 180,E1 -711.939,E2 -711.939} C_VEL
LIN {X 0,Y 601.426,Z 182.883,A -85,B 0,C 180,E1 -714.636,E2 -714.636} C_VEL
LIN {X 0,Y 601.428,Z 182.875,A -85,B 0,C 180,E1 -717.321,E2 -717.321} C_VEL
LIN {X 0,Y 601.432,Z 182.88,A -85,B 0,C 180,E1 -720,E2 -720} C_VEL
LIN {X 0,Y 601.442,Z 182.877,A -85,B 0,C 180,E1 -722.679,E2 -722.679} C_VEL
LIN {X 0,Y 601.417,Z 182.877,A -85,B 0,C 180,E1 -725.364,E2 -725.364} C_VEL
LIN {X 0,Y 601.435,Z 182.884,A -85,B 0,C 180,E1 -728.061,E2 -728.061} C_VEL
LIN {X 0,Y 601.424,Z 182.876,A -85,B 0,C 180,E1 -731.016,E2 -731.016} C_VEL
LIN {X 0,Y 601.412,Z 182.88,A -85,B 0,C 180,E1 -733.516,E2 -733.516} C_VEL
LIN {X 0,Y 601.436,Z 182.878,A -85,B 0,C 180,E1 -736.287,E2 -736.287} C_VEL
LIN {X 0,Y 601.411,Z 182.878,A -85,B 0,C 180,E1 -739.099,E2 -739.099} C_VEL
LIN {X 0,Y 601.403,Z 182.881,A -85,B 0,C 180,E1 -741.239,E2 -741.239} C_VEL
LIN {X 0,Y 601.45,Z 182.876,A -85,B 0,C 180,E1 -744.141,E2 -744.141} C_VEL
LIN {X 0,Y 601.446,Z 182.875,A -85,B 0,C 180,E1 -747.111,E2 -747.111} C_VEL
LIN {X 0,Y 601.417,Z 182.884,A -85,B 0,C 180,E1 -749.393,E2 -749.393} C_VEL
LIN {X 0,Y 601.407,Z 182.884,A -85,B 0,C 180,E1 -751.726,E2 -751.726} C_VEL
LIN {X 0,Y 601.426,Z 182.877,A -85,B 0,C 180,E1 -754.118,E2 -754.118} C_VEL
LIN {X 0,Y 601.431,Z 182.885,A -85,B 0,C 180,E1 -757.383,E2 -757.383} C_VEL
LIN {X 0,Y 601.403,Z 182.879,A -85,B 0,C 180,E1 -759.995,E2 -759.995} C_VEL
LIN {X 0,Y 601.408,Z 182.88,A -85,B 0,C 180,E1 -762.67,E2 -762.67} C_VEL
LIN {X 0,Y 601.392,Z 182.885,A -85,B 0,C 180,E1 -765.48,E2 -765.48} C_VEL
LIN {X 0,Y 601.421,Z 182.878,A -85,B 0,C 180,E1 -768.407,E2 -768.407} C_VEL
LIN {X 0,Y 601.428,Z 182.884,A -85,B 0,C 180,E1 -770.876,E2 -770.876} C_VEL
LIN {X 0,Y 601.398,Z 182.882,A -85,B 0,C 180,E1 -773.417,E2 -773.417} C_VEL
LIN {X 0,Y 601.426,Z 182.876,A -85,B 0,C 180,E1 -776.065,E2 -776.065} C_VEL
LIN {X 0,Y 601.412,Z 182.884,A -85,B 0,C 180,E1 -779.058,E2 -779.058} C_VEL
LIN {X 0,Y 601.398,Z 182.882,A -85,B 0,C 180,E1 -781.372,E2 -781.372} C_VEL
LIN {X 0,Y 601.424,Z 182.985,A -85,B 0,C 180,E1 -783.088,E2 -783.088} C_VEL
LIN {X 0,Y 602.147,Z 186.159,A -85,B 0,C 180,E1 -783.392,E2 -783.392} C_VEL
LIN {X 0,Y 602.059,Z 215.971,A -85,B 0,C 180,E1 -785.886,E2 -785.886} C_VEL
LIN {X 0,Y 602.02,Z 235.357,A -85,B 0,C 180,E1 -787.461,E2 -787.461} C_VEL
LIN {X 0,Y 602.358,Z 238.935,A -85,B 0,C 180,E1 -787.52,E2 -787.52} C_VEL
LIN {X 0,Y 602.111,Z 440.97,A -85,B 0,C 180,E1 -790.06,E2 -790.06} C_VEL
LIN {X 0,Y 602.074,Z 457.193,A -85,B 0,C 180,E1 -790.392,E2 -790.392} C_VEL
LIN {X 0,Y 602.01,Z 473.953,A -85,B 0,C 180,E1 -790.877,E2 -790.877} C_VEL
LIN {X 0,Y 601.915,Z 489.245,A -85,B 0,C 180,E1 -791.453,E2 -791.453} C_VEL
LIN {X 0,Y 601.869,Z 504.022,A -85,B 0,C 180,E1 -792.151,E2 -792.151} C_VEL
LIN {X 0,Y 601.767,Z 517.85,A -85,B 0,C 180,E1 -792.937,E2 -792.937} C_VEL
LIN {X 0,Y 601.695,Z 532.055,A -85,B 0,C 180,E1 -793.895,E2 -793.895} C_VEL
LIN {X 0,Y 601.592,Z 545.131,A -85,B 0,C 180,E1 -794.934,E2 -794.934} C_VEL
LIN {X 0,Y 601.555,Z 557.68,A -85,B 0,C 180,E1 -796.108,E2 -796.108} C_VEL
LIN {X 0,Y 601.472,Z 568.914,A -85,B 0,C 180,E1 -797.345,E2 -797.345} C_VEL
LIN {X 0,Y 601.427,Z 579.289,A -85,B 0,C 180,E1 -798.691,E2 -798.691} C_VEL
LIN {X 0,Y 601.388,Z 588.274,A -85,B 0,C 180,E1 -800.075,E2 -800.075} C_VEL
LIN {X 0,Y 601.364,Z 596.488,A -85,B 0,C 180,E1 -801.6,E2 -801.6} C_VEL
LIN {X 0,Y 601.361,Z 602.469,A -85,B 0,C 180,E1 -802.952,E2 -802.952} C_VEL
LIN {X 0,Y 601.346,Z 608.246,A -85,B 0,C 180,E1 -804.635,E2 -804.635} C_VEL
LIN {X 0,Y 601.339,Z 611.634,A -85,B 0,C 180,E1 -805.979,E2 -805.979} C_VEL
LIN {X 0,Y 601.311,Z 614.087,A -85,B 0,C 180,E1 -807.321,E2 -807.321} C_VEL
LIN {X 0,Y 601.341,Z 615.478,A -85,B 0,C 180,E1 -808.661,E2 -808.661} C_VEL
LIN {X 0,Y 601.33,Z 616,A -85,B 0,C 180,E1 -810,E2 -810} C_VEL
LIN {X 0,Y 601.34,Z 615.477,A -85,B 0,C 180,E1 -811.34,E2 -811.34} C_VEL
LIN {X 0,Y 601.311,Z 614.086,A -85,B 0,C 180,E1 -812.68,E2 -812.68} C_VEL
LIN {X 0,Y 601.339,Z 611.633,A -85,B 0,C 180,E1 -814.021,E2 -814.021} C_VEL
LIN {X 0,Y 601.346,Z 608.246,A -85,B 0,C 180,E1 -815.365,E2 -815.365} C_VEL
LIN {X 0,Y 601.362,Z 602.468,A -85,B 0,C 180,E1 -817.049,E2 -817.049} C_VEL
LIN {X 0,Y 601.376,Z 594.857,A -85,B 0,C 180,E1 -818.739,E2 -818.739} C_VEL
LIN {X 0,Y 601.41,Z 586.246,A -85,B 0,C 180,E1 -820.266,E2 -820.266} C_VEL
LIN {X 0,Y 601.43,Z 576.969,A -85,B 0,C 180,E1 -821.629,E2 -821.629} C_VEL
LIN {X 0,Y 601.479,Z 567.422,A -85,B 0,C 180,E1 -822.827,E2 -822.827} C_VEL
LIN {X 0,Y 601.545,Z 556.616,A -85,B 0,C 180,E1 -823.997,E2 -823.997} C_VEL
LIN {X 0,Y 601.606,Z 544.143,A -85,B 0,C 180,E1 -825.152,E2 -825.152} C_VEL
LIN {X 0,Y 601.707,Z 530.885,A -85,B 0,C 180,E1 -826.192,E2 -826.192} C_VEL
LIN {X 0,Y 601.764,Z 516.432,A -85,B 0,C 180,E1 -827.151,E2 -827.151} C_VEL
LIN {X 0,Y 601.864,Z 502.264,A -85,B 0,C 180,E1 -827.938,E2 -827.938} C_VEL
LIN {X 0,Y 601.942,Z 487.912,A -85,B 0,C 180,E1 -828.604,E2 -828.604} C_VEL
LIN {X 0,Y 602.011,Z 471.348,A -85,B 0,C 180,E1 -829.212,E2 -829.212} C_VEL
LIN {X 0,Y 602.09,Z 455.352,A -85,B 0,C 180,E1 -829.653,E2 -829.653} C_VEL
LIN {X 0,Y 602.118,Z 439.438,A -85,B 0,C 180,E1 -829.963,E2 -829.963} C_VEL
LIN {X 0,Y 602.321,Z 237.16,A -85,B 0,C 180,E1 -832.504,E2 -832.504} C_VEL
LIN {X 0,Y 601.968,Z 234.827,A -85,B 0,C 180,E1 -832.563,E2 -832.563} C_VEL
LIN {X 0,Y 602.085,Z 203.821,A -85,B 0,C 180,E1 -835.125,E2 -835.125} C_VEL
LIN {X 0,Y 602.168,Z 186.154,A -85,B 0,C 180,E1 -836.608,E2 -836.608} C_VEL
LIN {X 0,Y 601.398,Z 182.887,A -85,B 0,C 180,E1 -836.926,E2 -836.926} C_VEL
LIN {X 0,Y 601.398,Z 182.888,A -85,B 0,C 180,E1 -839.394,E2 -839.394} C_VEL
LIN {X 0,Y 601.389,Z 182.883,A -85,B 0,C 180,E1 -841.727,E2 -841.727} C_VEL
LIN {X 0,Y 601.415,Z 182.877,A -85,B 0,C 180,E1 -844.119,E2 -844.119} C_VEL
LIN {X 0,Y 601.391,Z 182.882,A -85,B 0,C 180,E1 -846.583,E2 -846.583} C_VEL
LIN {X 0,Y 601.434,Z 182.878,A -85,B 0,C 180,E1 -849.535,E2 -849.535} C_VEL
LIN {X 0,Y 601.41,Z 182.878,A -85,B 0,C 180,E1 -851.766,E2 -851.766} C_VEL
LIN {X 0,Y 601.394,Z 182.882,A -85,B 0,C 180,E1 -854.532,E2 -854.532} C_VEL
LIN {X 0,Y 601.408,Z 182.881,A -85,B 0,C 180,E1 -857.409,E2 -857.409} C_VEL
LIN {X 0,Y 601.395,Z 182.879,A -85,B 0,C 180,E1 -860.004,E2 -860.004} C_VEL
LIN {X 0,Y 601.432,Z 182.88,A -85,B 0,C 180,E1 -862.618,E2 -862.618} C_VEL
LIN {X 0,Y 601.416,Z 182.877,A -85,B 0,C 180,E1 -865.881,E2 -865.881} C_VEL
LIN {X 0,Y 601.436,Z 182.88,A -85,B 0,C 180,E1 -868.542,E2 -868.542} C_VEL
LIN {X 0,Y 601.428,Z 182.877,A -85,B 0,C 180,E1 -871.373,E2 -871.373} C_VEL
LIN {X 0,Y 601.391,Z 182.879,A -85,B 0,C 180,E1 -873.636,E2 -873.636} C_VEL
LIN {X 0,Y 601.412,Z 182.886,A -85,B 0,C 180,E1 -876.589,E2 -876.589} C_VEL
LIN {X 0,Y 601.419,Z 182.876,A -85,B 0,C 180,E1 -879.478,E2 -879.478} C_VEL
LIN {X 0,Y 601.388,Z 182.885,A -85,B 0,C 180,E1 -882.311,E2 -882.311} C_VEL
LIN {X 0,Y 601.423,Z 182.877,A -85,B 0,C 180,E1 -885.103,E2 -885.103} C_VEL
LIN {X 0,Y 601.405,Z 182.878,A -85,B 0,C 180,E1 -887.857,E2 -887.857} C_VEL
LIN {X 0,Y 601.414,Z 182.885,A -85,B 0,C 180,E1 -890.584,E2 -890.584} C_VEL
LIN {X 0,Y 601.427,Z 182.875,A -85,B 0,C 180,E1 -893.345,E2 -893.345} C_VEL
LIN {X 0,Y 601.394,Z 182.883,A -85,B 0,C 180,E1 -895.979,E2 -895.979} C_VEL
LIN {X 0,Y 601.425,Z 182.879,A -85,B 0,C 180,E1 -898.661,E2 -898.661} C_VEL
LIN {X 0,Y 601.41,Z 182.877,A -85,B 0,C 180,E1 -901.339,E2 -901.339} C_VEL
LIN {X 0,Y 601.419,Z 182.876,A -85,B 0,C 180,E1 -903.35,E2 -903.35} C_VEL
LIN {X 0,Y 601.403,Z 182.885,A -85,B 0,C 180,E1 -906.037,E2 -906.037} C_VEL
LIN {X 0,Y 601.412,Z 182.879,A -85,B 0,C 180,E1 -908.738,E2 -908.738} C_VEL
LIN {X 0,Y 601.429,Z 182.876,A -85,B 0,C 180,E1 -911.458,E2 -911.458} C_VEL
LIN {X 0,Y 601.405,Z 182.883,A -85,B 0,C 180,E1 -912.379,E2 -912.379} C_VEL
LIN {X 0,Y 600.74,Z 182.963,A -85,B 0,C 180,E1 -912.938,E2 -912.938} C_VEL
LIN {X 0,Y 597.889,Z 183.322,A -85,B 0,C 180,E1 -913.846,E2 -913.846} C_VEL
LIN {X 0,Y 595.479,Z 183.619,A -85,B 0,C 180,E1 -914.576,E2 -914.576} C_VEL
LIN {X 0,Y 594.441,Z 183.746,A -85,B 0,C 180,E1 -915.14,E2 -915.14} C_VEL
LIN {X 0,Y 594.356,Z 183.757,A -85,B 0,C 180,E1 -915.331,E2 -915.331} C_VEL
LIN {X 0,Y 594.376,Z 183.762,A -85,B 0,C 180,E1 -917.904,E2 -917.904} C_VEL
LIN {X 0,Y 594.378,Z 183.753,A -85,B 0,C 180,E1 -920.917,E2 -920.917} C_VEL
LIN {X 0,Y 594.389,Z 183.759,A -85,B 0,C 180,E1 -923.704,E2 -923.704} C_VEL
LIN {X 0,Y 594.38,Z 183.753,A -85,B 0,C 180,E1 -926.7,E2 -926.7} C_VEL
LIN {X 0,Y 594.379,Z 183.754,A -85,B 0,C 180,E1 -928.998,E2 -928.998} C_VEL
LIN {X 0,Y 594.375,Z 183.762,A -85,B 0,C 180,E1 -931.643,E2 -931.643} C_VEL
LIN {X 0,Y 594.391,Z 183.752,A -85,B 0,C 180,E1 -934.579,E2 -934.579} C_VEL
LIN {X 0,Y 594.381,Z 183.755,A -85,B 0,C 180,E1 -937.087,E2 -937.087} C_VEL
LIN {X 0,Y 594.356,Z 183.764,A -85,B 0,C 180,E1 -939.773,E2 -939.773} C_VEL
LIN {X 0,Y 594.366,Z 183.755,A -85,B 0,C 180,E1 -942.375,E2 -942.375} C_VEL
LIN {X 0,Y 594.361,Z 183.76,A -85,B 0,C 180,E1 -945.191,E2 -945.191} C_VEL
LIN {X 0,Y 594.379,Z 183.754,A -85,B 0,C 180,E1 -948.152,E2 -948.152} C_VEL
LIN {X 0,Y 594.375,Z 183.76,A -85,B 0,C 180,E1 -951.195,E2 -951.195} C_VEL
LIN {X 0,Y 594.35,Z 183.76,A -85,B 0,C 180,E1 -953.756,E2 -953.756} C_VEL
LIN {X 0,Y 594.378,Z 183.753,A -85,B 0,C 180,E1 -956.239,E2 -956.239} C_VEL
LIN {X 0,Y 594.378,Z 183.754,A -85,B 0,C 180,E1 -958.65,E2 -958.65} C_VEL
LIN {X 0,Y 594.383,Z 183.76,A -85,B 0,C 180,E1 -961.042,E2 -961.042} C_VEL
LIN {X 0,Y 594.391,Z 183.752,A -85,B 0,C 180,E1 -963.976,E2 -963.976} C_VEL
LIN {X 0,Y 594.387,Z 183.752,A -85,B 0,C 180,E1 -966.296,E2 -966.296} C_VEL
LIN {X 0,Y 594.4,Z 183.758,A -85,B 0,C 180,E1 -969.224,E2 -969.224} C_VEL
LIN {X 0,Y 594.353,Z 183.756,A -85,B 0,C 180,E1 -972.095,E2 -972.095} C_VEL
LIN {X 0,Y 594.364,Z 183.756,A -85,B 0,C 180,E1 -974.219,E2 -974.219} C_VEL
LIN {X 0,Y 594.384,Z 183.752,A -85,B 0,C 180,E1 -976.321,E2 -976.321} C_VEL
LIN {X 0,Y 594.371,Z 183.763,A -85,B 0,C 180,E1 -979.095,E2 -979.095} C_VEL
LIN {X 0,Y 594.411,Z 183.75,A -85,B 0,C 180,E1 -981.843,E2 -981.843} C_VEL
LIN {X 0,Y 594.4,Z 183.756,A -85,B 0,C 180,E1 -984.572,E2 -984.572} C_VEL
LIN {X 0,Y 594.395,Z 183.755,A -85,B 0,C 180,E1 -987.289,E2 -987.289} C_VEL
LIN {X 0,Y 594.414,Z 183.752,A -85,B 0,C 180,E1 -990,E2 -990} C_VEL
LIN {X 0,Y 594.416,Z 183.763,A -85,B 0,C 180,E1 -991.101,E2 -991.101} C_VEL
LIN {X 0,Y 595.216,Z 187.791,A -85,B 0,C 180,E1 -991.522,E2 -991.522} C_VEL
LIN {X 0,Y 595.101,Z 205.926,A -85,B 0,C 180,E1 -993.237,E2 -993.237} C_VEL
LIN {X 0,Y 595.792,Z 210.057,A -85,B 0,C 180,E1 -993.318,E2 -993.318} C_VEL
LIN {X 0,Y 595.449,Z 411.789,A -85,B 0,C 180,E1 -995.885,E2 -995.885} C_VEL
LIN {X 0,Y 595.372,Z 428.505,A -85,B 0,C 180,E1 -996.238,E2 -996.238} C_VEL
LIN {X 0,Y 595.282,Z 445.135,A -85,B 0,C 180,E1 -996.737,E2 -996.737} C_VEL
LIN {X 0,Y 595.149,Z 460.6,A -85,B 0,C 180,E1 -997.34,E2 -997.34} C_VEL
LIN {X 0,Y 595.045,Z 475.53,A -85,B 0,C 180,E1 -998.062,E2 -998.062} C_VEL
LIN {X 0,Y 594.895,Z 490.095,A -85,B 0,C 180,E1 -998.92,E2 -998.92} C_VEL
LIN {X 0,Y 594.767,Z 503.612,A -85,B 0,C 180,E1 -999.865,E2 -999.865} C_VEL
LIN {X 0,Y 594.632,Z 517.495,A -85,B 0,C 180,E1 -1001.012,E2 -1001.012} C_VEL
LIN {X 0,Y 594.535,Z 528.86,A -85,B 0,C 180,E1 -1002.112,E2 -1002.112} C_VEL
LIN {X 0,Y 594.471,Z 539.67,A -85,B 0,C 180,E1 -1003.328,E2 -1003.328} C_VEL
LIN {X 0,Y 594.387,Z 550.191,A -85,B 0,C 180,E1 -1004.727,E2 -1004.727} C_VEL
LIN {X 0,Y 594.331,Z 559.064,A -85,B 0,C 180,E1 -1006.134,E2 -1006.134} C_VEL
LIN {X 0,Y 594.309,Z 566.517,A -85,B 0,C 180,E1 -1007.55,E2 -1007.55} C_VEL
LIN {X 0,Y 594.288,Z 572.43,A -85,B 0,C 180,E1 -1008.903,E2 -1008.903} C_VEL
LIN {X 0,Y 594.267,Z 577.63,A -85,B 0,C 180,E1 -1010.418,E2 -1010.418} C_VEL
LIN {X 0,Y 594.227,Z 580.609,A -85,B 0,C 180,E1 -1011.508,E2 -1011.508} C_VEL
LIN {X 0,Y 594.208,Z 583.501,A -85,B 0,C 180,E1 -1012.973,E2 -1012.973} C_VEL
LIN {X 0,Y 594.205,Z 585.315,A -85,B 0,C 180,E1 -1014.454,E2 -1014.454} C_VEL
LIN {X 0,Y 594.224,Z 585.994,A -85,B 0,C 180,E1 -1015.991,E2 -1015.991} C_VEL
LIN {X 0,Y 594.246,Z 585.408,A -85,B 0,C 180,E1 -1017.501,E2 -1017.501} C_VEL
LIN {X 0,Y 594.245,Z 583.683,A -85,B 0,C 180,E1 -1019.005,E2 -1019.005} C_VEL
LIN {X 0,Y 594.23,Z 580.647,A -85,B 0,C 180,E1 -1020.568,E2 -1020.568} C_VEL
LIN {X 0,Y 594.255,Z 577.78,A -85,B 0,C 180,E1 -1021.624,E2 -1021.624} C_VEL
LIN {X 0,Y 594.256,Z 573.283,A -85,B 0,C 180,E1 -1022.957,E2 -1022.957} C_VEL
LIN {X 0,Y 594.313,Z 567.517,A -85,B 0,C 180,E1 -1024.328,E2 -1024.328} C_VEL
LIN {X 0,Y 594.321,Z 559.822,A -85,B 0,C 180,E1 -1025.827,E2 -1025.827} C_VEL
LIN {X 0,Y 594.349,Z 552.039,A -85,B 0,C 180,E1 -1027.088,E2 -1027.088} C_VEL
LIN {X 0,Y 594.408,Z 542.776,A -85,B 0,C 180,E1 -1028.369,E2 -1028.369} C_VEL
LIN {X 0,Y 594.496,Z 531.749,A -85,B 0,C 180,E1 -1029.67,E2 -1029.67} C_VEL
LIN {X 0,Y 594.61,Z 520.039,A -85,B 0,C 180,E1 -1030.848,E2 -1030.848} C_VEL
LIN {X 0,Y 594.729,Z 506.837,A -85,B 0,C 180,E1 -1031.98,E2 -1031.98} C_VEL
LIN {X 0,Y 594.872,Z 492.545,A -85,B 0,C 180,E1 -1033.014,E2 -1033.014} C_VEL
LIN {X 0,Y 594.997,Z 477.798,A -85,B 0,C 180,E1 -1033.903,E2 -1033.903} C_VEL
LIN {X 0,Y 595.112,Z 463.053,A -85,B 0,C 180,E1 -1034.64,E2 -1034.64} C_VEL
LIN {X 0,Y 595.256,Z 447.14,A -85,B 0,C 180,E1 -1035.284,E2 -1035.284} C_VEL
LIN {X 0,Y 595.352,Z 430.952,A -85,B 0,C 180,E1 -1035.79,E2 -1035.79} C_VEL
LIN {X 0,Y 595.461,Z 413.859,A -85,B 0,C 180,E1 -1036.17,E2 -1036.17} C_VEL
LIN {X 0,Y 595.511,Z 381.718,A -85,B 0,C 180,E1 -1036.602,E2 -1036.602} C_VEL
LIN {X 0,Y 595.742,Z 209.83,A -85,B 0,C 180,E1 -1038.777,E2 -1038.777} C_VEL
LIN {X 0,Y 595.038,Z 205.806,A -85,B 0,C 180,E1 -1038.864,E2 -1038.864} C_VEL
LIN {X 0,Y 595.147,Z 187.481,A -85,B 0,C 180,E1 -1040.601,E2 -1040.601} C_VEL
LIN {X 0,Y 594.327,Z 183.769,A -85,B 0,C 180,E1 -1041,E2 -1041} C_VEL
LIN {X 0,Y 594.334,Z 183.763,A -85,B 0,C 180,E1 -1043.754,E2 -1043.754} C_VEL
LIN {X 0,Y 594.341,Z 183.758,A -85,B 0,C 180,E1 -1046.236,E2 -1046.236} C_VEL
LIN {X 0,Y 594.351,Z 183.761,A -85,B 0,C 180,E1 -1048.649,E2 -1048.649} C_VEL
LIN {X 0,Y 594.373,Z 183.764,A -85,B 0,C 180,E1 -1051.042,E2 -1051.042} C_VEL
LIN {X 0,Y 594.34,Z 183.759,A -85,B 0,C 180,E1 -1053.984,E2 -1053.984} C_VEL
LIN {X 0,Y 594.352,Z 183.758,A -85,B 0,C 180,E1 -1056.294,E2 -1056.294} C_VEL
LIN {X 0,Y 594.394,Z 183.756,A -85,B 0,C 180,E1 -1059.224,E2 -1059.224} C_VEL
LIN {X 0,Y 594.332,Z 183.76,A -85,B 0,C 180,E1 -1062.094,E2 -1062.094} C_VEL
LIN {X 0,Y 594.351,Z 183.759,A -85,B 0,C 180,E1 -1064.219,E2 -1064.219} C_VEL
LIN {X 0,Y 594.364,Z 183.76,A -85,B 0,C 180,E1 -1066.321,E2 -1066.321} C_VEL
LIN {X 0,Y 594.369,Z 183.757,A -85,B 0,C 180,E1 -1069.095,E2 -1069.095} C_VEL
LIN {X 0,Y 594.368,Z 183.756,A -85,B 0,C 180,E1 -1071.843,E2 -1071.843} C_VEL
LIN {X 0,Y 594.388,Z 183.761,A -85,B 0,C 180,E1 -1074.572,E2 -1074.572} C_VEL
LIN {X 0,Y 594.396,Z 183.751,A -85,B 0,C 180,E1 -1077.289,E2 -1077.289} C_VEL
LIN {X 0,Y 594.401,Z 183.756,A -85,B 0,C 180,E1 -1080,E2 -1080} C_VEL
LIN {X 0,Y 594.407,Z 183.753,A -85,B 0,C 180,E1 -1082.711,E2 -1082.711} C_VEL
LIN {X 0,Y 594.381,Z 183.754,A -85,B 0,C 180,E1 -1085.428,E2 -1085.428} C_VEL
LIN {X 0,Y 594.411,Z 183.759,A -85,B 0,C 180,E1 -1088.157,E2 -1088.157} C_VEL
LIN {X 0,Y 594.387,Z 183.752,A -85,B 0,C 180,E1 -1091.077,E2 -1091.077} C_VEL
LIN {X 0,Y 594.377,Z 183.759,A -85,B 0,C 180,E1 -1093.679,E2 -1093.679} C_VEL
LIN {X 0,Y 594.389,Z 183.752,A -85,B 0,C 180,E1 -1096.72,E2 -1096.72} C_VEL
LIN {X 0,Y 594.361,Z 183.758,A -85,B 0,C 180,E1 -1099.335,E2 -1099.335} C_VEL
LIN {X 0,Y 594.362,Z 183.762,A -85,B 0,C 180,E1 -1101.503,E2 -1101.503} C_VEL
LIN {X 0,Y 594.382,Z 183.754,A -85,B 0,C 180,E1 -1104.446,E2 -1104.446} C_VEL
LIN {X 0,Y 594.381,Z 183.753,A -85,B 0,C 180,E1 -1106.7,E2 -1106.7} C_VEL
LIN {X 0,Y 594.378,Z 183.756,A -85,B 0,C 180,E1 -1108.999,E2 -1108.999} C_VEL
LIN {X 0,Y 594.386,Z 183.761,A -85,B 0,C 180,E1 -1111.646,E2 -1111.646} C_VEL
LIN {X 0,Y 594.391,Z 183.753,A -85,B 0,C 180,E1 -1114.579,E2 -1114.579} C_VEL
LIN {X 0,Y 594.383,Z 183.759,A -85,B 0,C 180,E1 -1117.609,E2 -1117.609} C_VEL
LIN {X 0,Y 594.365,Z 183.757,A -85,B 0,C 180,E1 -1120.567,E2 -1120.567} C_VEL
LIN {X 0,Y 594.362,Z 183.765,A -85,B 0,C 180,E1 -1123.3,E2 -1123.3} C_VEL
LIN {X 0,Y 594.354,Z 183.757,A -85,B 0,C 180,E1 -1126.162,E2 -1126.162} C_VEL
LIN {X 0,Y 594.378,Z 183.757,A -85,B 0,C 180,E1 -1128.537,E2 -1128.537} C_VEL
LIN {X 0,Y 594.372,Z 183.76,A -85,B 0,C 180,E1 -1131.297,E2 -1131.297} C_VEL
LIN {X 0,Y 594.344,Z 183.759,A -85,B 0,C 180,E1 -1133.756,E2 -1133.756} C_VEL
LIN {X 0,Y 594.372,Z 183.756,A -85,B 0,C 180,E1 -1136.239,E2 -1136.239} C_VEL
LIN {X 0,Y 594.383,Z 183.761,A -85,B 0,C 180,E1 -1138.651,E2 -1138.651} C_VEL
LIN {X 0,Y 594.369,Z 183.762,A -85,B 0,C 180,E1 -1141.044,E2 -1141.044} C_VEL
LIN {X 0,Y 594.404,Z 183.951,A -85,B 0,C 180,E1 -1142.827,E2 -1142.827} C_VEL
LIN {X 0,Y 595.52,Z 188.368,A -85,B 0,C 180,E1 -1143.261,E2 -1143.261} C_VEL
LIN {X 0,Y 595.305,Z 220.388,A -85,B 0,C 180,E1 -1145.965,E2 -1145.965} C_VEL
LIN {X 0,Y 595.189,Z 234.994,A -85,B 0,C 180,E1 -1147.18,E2 -1147.18} C_VEL
LIN {X 0,Y 595.807,Z 238.681,A -85,B 0,C 180,E1 -1147.256,E2 -1147.256} C_VEL
LIN {X 0,Y 595.439,Z 442.458,A -85,B 0,C 180,E1 -1149.849,E2 -1149.849} C_VEL
LIN {X 0,Y 595.405,Z 459.02,A -85,B 0,C 180,E1 -1150.208,E2 -1150.208} C_VEL
LIN {X 0,Y 595.286,Z 475.249,A -85,B 0,C 180,E1 -1150.697,E2 -1150.697} C_VEL
LIN {X 0,Y 595.121,Z 491.896,A -85,B 0,C 180,E1 -1151.353,E2 -1151.353} C_VEL
LIN {X 0,Y 595.004,Z 507.316,A -85,B 0,C 180,E1 -1152.116,E2 -1152.116} C_VEL
LIN {X 0,Y 594.896,Z 521.144,A -85,B 0,C 180,E1 -1152.94,E2 -1152.94} C_VEL
LIN {X 0,Y 594.764,Z 534.38,A -85,B 0,C 180,E1 -1153.878,E2 -1153.878} C_VEL
LIN {X 0,Y 594.634,Z 547.074,A -85,B 0,C 180,E1 -1154.929,E2 -1154.929} C_VEL
LIN {X 0,Y 594.553,Z 558.977,A -85,B 0,C 180,E1 -1156.08,E2 -1156.08} C_VEL
LIN {X 0,Y 594.461,Z 570.335,A -85,B 0,C 180,E1 -1157.367,E2 -1157.367} C_VEL
LIN {X 0,Y 594.385,Z 580.629,A -85,B 0,C 180,E1 -1158.743,E2 -1158.743} C_VEL
LIN {X 0,Y 594.337,Z 589.287,A -85,B 0,C 180,E1 -1160.128,E2 -1160.128} C_VEL
LIN {X 0,Y 594.295,Z 596.488,A -85,B 0,C 180,E1 -1161.5,E2 -1161.5} C_VEL
LIN {X 0,Y 594.284,Z 602.469,A -85,B 0,C 180,E1 -1162.867,E2 -1162.867} C_VEL
LIN {X 0,Y 594.264,Z 608.247,A -85,B 0,C 180,E1 -1164.571,E2 -1164.571} C_VEL
LIN {X 0,Y 594.252,Z 611.635,A -85,B 0,C 180,E1 -1165.931,E2 -1165.931} C_VEL
LIN {X 0,Y 594.213,Z 614.087,A -85,B 0,C 180,E1 -1167.289,E2 -1167.289} C_VEL
LIN {X 0,Y 594.24,Z 615.478,A -85,B 0,C 180,E1 -1168.645,E2 -1168.645} C_VEL
LIN {X 0,Y 594.231,Z 616,A -85,B 0,C 180,E1 -1170,E2 -1170} C_VEL
LIN {X 0,Y 594.24,Z 615.478,A -85,B 0,C 180,E1 -1171.356,E2 -1171.356} C_VEL
LIN {X 0,Y 594.213,Z 614.087,A -85,B 0,C 180,E1 -1172.712,E2 -1172.712} C_VEL
LIN {X 0,Y 594.252,Z 611.633,A -85,B 0,C 180,E1 -1174.069,E2 -1174.069} C_VEL
LIN {X 0,Y 594.281,Z 607.185,A -85,B 0,C 180,E1 -1175.769,E2 -1175.769} C_VEL
LIN {X 0,Y 594.284,Z 602.468,A -85,B 0,C 180,E1 -1177.133,E2 -1177.133} C_VEL
LIN {X 0,Y 594.318,Z 594.857,A -85,B 0,C 180,E1 -1178.843,E2 -1178.843} C_VEL
LIN {X 0,Y 594.354,Z 586.247,A -85,B 0,C 180,E1 -1180.389,E2 -1180.389} C_VEL
LIN {X 0,Y 594.407,Z 576.97,A -85,B 0,C 180,E1 -1181.768,E2 -1181.768} C_VEL
LIN {X 0,Y 594.469,Z 567.423,A -85,B 0,C 180,E1 -1182.981,E2 -1182.981} C_VEL
LIN {X 0,Y 594.539,Z 555.949,A -85,B 0,C 180,E1 -1184.231,E2 -1184.231} C_VEL
LIN {X 0,Y 594.678,Z 544.143,A -85,B 0,C 180,E1 -1185.333,E2 -1185.333} C_VEL
LIN {X 0,Y 594.809,Z 530.882,A -85,B 0,C 180,E1 -1186.385,E2 -1186.385} C_VEL
LIN {X 0,Y 594.924,Z 516.435,A -85,B 0,C 180,E1 -1187.355,E2 -1187.355} C_VEL
LIN {X 0,Y 595.046,Z 502.268,A -85,B 0,C 180,E1 -1188.15,E2 -1188.15} C_VEL
LIN {X 0,Y 595.199,Z 487.114,A -85,B 0,C 180,E1 -1188.854,E2 -1188.854} C_VEL
LIN {X 0,Y 595.279,Z 471.347,A -85,B 0,C 180,E1 -1189.438,E2 -1189.438} C_VEL
LIN {X 0,Y 595.382,Z 455.354,A -85,B 0,C 180,E1 -1189.883,E2 -1189.883} C_VEL
LIN {X 0,Y 595.466,Z 439.437,A -85,B 0,C 180,E1 -1190.195,E2 -1190.195} C_VEL
LIN {X 0,Y 595.784,Z 238.468,A -85,B 0,C 180,E1 -1192.748,E2 -1192.748} C_VEL
LIN {X 0,Y 595.217,Z 235.027,A -85,B 0,C 180,E1 -1192.816,E2 -1192.816} C_VEL
LIN {X 0,Y 595.397,Z 203.821,A -85,B 0,C 180,E1 -1195.427,E2 -1195.427} C_VEL
LIN {X 0,Y 595.519,Z 188.363,A -85,B 0,C 180,E1 -1196.739,E2 -1196.739} C_VEL
LIN {X 0,Y 594.379,Z 183.764,A -85,B 0,C 180,E1 -1197.198,E2 -1197.198} C_VEL
LIN {X 0,Y 594.355,Z 183.76,A -85,B 0,C 180,E1 -1199.777,E2 -1199.777} C_VEL
LIN {X 0,Y 594.345,Z 183.757,A -85,B 0,C 180,E1 -1202.148,E2 -1202.148} C_VEL
LIN {X 0,Y 594.367,Z 183.757,A -85,B 0,C 180,E1 -1204.581,E2 -1204.581} C_VEL
LIN {X 0,Y 594.383,Z 183.756,A -85,B 0,C 180,E1 -1207.608,E2 -1207.608} C_VEL
LIN {X 0,Y 594.357,Z 183.758,A -85,B 0,C 180,E1 -1210.568,E2 -1210.568} C_VEL
LIN {X 0,Y 594.357,Z 183.762,A -85,B 0,C 180,E1 -1213.3,E2 -1213.3} C_VEL
LIN {X 0,Y 594.339,Z 183.758,A -85,B 0,C 180,E1 -1216.163,E2 -1216.163} C_VEL
LIN {X 0,Y 594.369,Z 183.758,A -85,B 0,C 180,E1 -1218.535,E2 -1218.535} C_VEL
LIN {X 0,Y 594.369,Z 183.759,A -85,B 0,C 180,E1 -1221.297,E2 -1221.297} C_VEL
LIN {X 0,Y 594.345,Z 183.757,A -85,B 0,C 180,E1 -1223.755,E2 -1223.755} C_VEL
LIN {X 0,Y 594.36,Z 183.757,A -85,B 0,C 180,E1 -1226.238,E2 -1226.238} C_VEL
LIN {X 0,Y 594.383,Z 183.76,A -85,B 0,C 180,E1 -1228.651,E2 -1228.651} C_VEL
LIN {X 0,Y 594.379,Z 183.759,A -85,B 0,C 180,E1 -1231.042,E2 -1231.042} C_VEL
LIN {X 0,Y 594.379,Z 183.754,A -85,B 0,C 180,E1 -1233.3,E2 -1233.3} C_VEL
LIN {X 0,Y 594.376,Z 183.757,A -85,B 0,C 180,E1 -1236.296,E2 -1236.296} C_VEL
LIN {X 0,Y 594.398,Z 183.752,A -85,B 0,C 180,E1 -1239.224,E2 -1239.224} C_VEL
LIN {X 0,Y 594.34,Z 183.76,A -85,B 0,C 180,E1 -1242.095,E2 -1242.095} C_VEL
LIN {X 0,Y 594.357,Z 183.761,A -85,B 0,C 180,E1 -1244.219,E2 -1244.219} C_VEL
LIN {X 0,Y 594.369,Z 183.761,A -85,B 0,C 180,E1 -1246.321,E2 -1246.321} C_VEL
LIN {X 0,Y 594.371,Z 183.754,A -85,B 0,C 180,E1 -1249.095,E2 -1249.095} C_VEL
LIN {X 0,Y 594.375,Z 183.756,A -85,B 0,C 180,E1 -1251.843,E2 -1251.843} C_VEL
LIN {X 0,Y 594.39,Z 183.757,A -85,B 0,C 180,E1 -1254.572,E2 -1254.572} C_VEL
LIN {X 0,Y 594.397,Z 183.748,A -85,B 0,C 180,E1 -1257.289,E2 -1257.289} C_VEL
LIN {X 0,Y 594.405,Z 183.755,A -85,B 0,C 180,E1 -1260,E2 -1260} C_VEL
LIN {X 0,Y 594.407,Z 183.752,A -85,B 0,C 180,E1 -1262.711,E2 -1262.711} C_VEL
LIN {X 0,Y 594.382,Z 183.752,A -85,B 0,C 180,E1 -1265.428,E2 -1265.428} C_VEL
LIN {X 0,Y 594.408,Z 183.76,A -85,B 0,C 180,E1 -1268.157,E2 -1268.157} C_VEL
LIN {X 0,Y 594.39,Z 183.751,A -85,B 0,C 180,E1 -1271.076,E2 -1271.076} C_VEL
LIN {X 0,Y 594.376,Z 183.757,A -85,B 0,C 180,E1 -1273.679,E2 -1273.679} C_VEL
LIN {X 0,Y 594.356,Z 183.757,A -85,B 0,C 180,E1 -1275.331,E2 -1275.331} C_VEL
LIN {X 0,Y 593.686,Z 183.848,A -85,B 0,C 180,E1 -1275.897,E2 -1275.897} C_VEL
LIN {X 0,Y 590.834,Z 184.205,A -85,B 0,C 180,E1 -1276.815,E2 -1276.815} C_VEL
LIN {X 0,Y 588.429,Z 184.504,A -85,B 0,C 180,E1 -1277.554,E2 -1277.554} C_VEL
LIN {X 0,Y 587.402,Z 184.628,A -85,B 0,C 180,E1 -1278.124,E2 -1278.124} C_VEL
LIN {X 0,Y 587.321,Z 184.635,A -85,B 0,C 180,E1 -1278.317,E2 -1278.317} C_VEL
LIN {X 0,Y 587.327,Z 184.631,A -85,B 0,C 180,E1 -1281.038,E2 -1281.038} C_VEL
LIN {X 0,Y 587.32,Z 184.634,A -85,B 0,C 180,E1 -1283.259,E2 -1283.259} C_VEL
LIN {X 0,Y 587.332,Z 184.634,A -85,B 0,C 180,E1 -1285.517,E2 -1285.517} C_VEL
LIN {X 0,Y 587.346,Z 184.64,A -85,B 0,C 180,E1 -1287.818,E2 -1287.818} C_VEL
LIN {X 0,Y 587.341,Z 184.63,A -85,B 0,C 180,E1 -1290.511,E2 -1290.511} C_VEL
LIN {X 0,Y 587.333,Z 184.635,A -85,B 0,C 180,E1 -1293.397,E2 -1293.397} C_VEL
LIN {X 0,Y 587.353,Z 184.635,A -85,B 0,C 180,E1 -1295.896,E2 -1295.896} C_VEL
LIN {X 0,Y 587.325,Z 184.631,A -85,B 0,C 180,E1 -1298.48,E2 -1298.48} C_VEL
LIN {X 0,Y 587.333,Z 184.635,A -85,B 0,C 180,E1 -1301.157,E2 -1301.157} C_VEL
LIN {X 0,Y 587.309,Z 184.635,A -85,B 0,C 180,E1 -1304.112,E2 -1304.112} C_VEL
LIN {X 0,Y 587.312,Z 184.636,A -85,B 0,C 180,E1 -1306.994,E2 -1306.994} C_VEL
LIN {X 0,Y 587.311,Z 184.639,A -85,B 0,C 180,E1 -1309.746,E2 -1309.746} C_VEL
LIN {X 0,Y 587.342,Z 184.63,A -85,B 0,C 180,E1 -1312.392,E2 -1312.392} C_VEL
LIN {X 0,Y 587.366,Z 184.63,A -85,B 0,C 180,E1 -1315.781,E2 -1315.781} C_VEL
LIN {X 0,Y 587.344,Z 184.629,A -85,B 0,C 180,E1 -1318.232,E2 -1318.232} C_VEL
LIN {X 0,Y 587.349,Z 184.633,A -85,B 0,C 180,E1 -1320.866,E2 -1320.866} C_VEL
LIN {X 0,Y 587.361,Z 184.629,A -85,B 0,C 180,E1 -1323.818,E2 -1323.818} C_VEL
LIN {X 0,Y 587.335,Z 184.63,A -85,B 0,C 180,E1 -1325.994,E2 -1325.994} C_VEL
LIN {X 0,Y 587.318,Z 184.633,A -85,B 0,C 180,E1 -1328.226,E2 -1328.226} C_VEL
LIN {X 0,Y 587.347,Z 184.637,A -85,B 0,C 180,E1 -1331.151,E2 -1331.151} C_VEL
LIN {X 0,Y 587.317,Z 184.633,A -85,B 0,C 180,E1 -1334.025,E2 -1334.025} C_VEL
LIN {X 0,Y 587.361,Z 184.626,A -85,B 0,C 180,E1 -1336.154,E2 -1336.154} C_VEL
LIN {X 0,Y 587.337,Z 184.64,A -85,B 0,C 180,E1 -1338.962,E2 -1338.962} C_VEL
LIN {X 0,Y 587.363,Z 184.628,A -85,B 0,C 180,E1 -1341.745,E2 -1341.745} C_VEL
LIN {X 0,Y 587.366,Z 184.631,A -85,B 0,C 180,E1 -1344.507,E2 -1344.507} C_VEL
LIN {X 0,Y 587.363,Z 184.632,A -85,B 0,C 180,E1 -1347.257,E2 -1347.257} C_VEL
LIN {X 0,Y 587.383,Z 184.629,A -85,B 0,C 180,E1 -1350,E2 -1350} C_VEL
LIN {X 0,Y 587.414,Z 184.744,A -85,B 0,C 180,E1 -1350.878,E2 -1350.878} C_VEL
LIN {X 0,Y 588.425,Z 189.324,A -85,B 0,C 180,E1 -1351.369,E2 -1351.369} C_VEL
LIN {X 0,Y 588.354,Z 206.168,A -85,B 0,C 180,E1 -1352.963,E2 -1352.963} C_VEL
LIN {X 0,Y 589.232,Z 210.441,A -85,B 0,C 180,E1 -1353.055,E2 -1353.055} C_VEL
LIN {X 0,Y 588.778,Z 412.049,A -85,B 0,C 180,E1 -1355.651,E2 -1355.651} C_VEL
LIN {X 0,Y 588.69,Z 429.029,A -85,B 0,C 180,E1 -1356.017,E2 -1356.017} C_VEL
LIN {X 0,Y 588.536,Z 445.339,A -85,B 0,C 180,E1 -1356.514,E2 -1356.514} C_VEL
LIN {X 0,Y 588.384,Z 460.869,A -85,B 0,C 180,E1 -1357.129,E2 -1357.129} C_VEL
LIN {X 0,Y 588.222,Z 476.453,A -85,B 0,C 180,E1 -1357.897,E2 -1357.897} C_VEL
LIN {X 0,Y 588.028,Z 490.896,A -85,B 0,C 180,E1 -1358.765,E2 -1358.765} C_VEL
LIN {X 0,Y 587.853,Z 504.292,A -85,B 0,C 180,E1 -1359.722,E2 -1359.722} C_VEL
LIN {X 0,Y 587.68,Z 517.785,A -85,B 0,C 180,E1 -1360.856,E2 -1360.856} C_VEL
LIN {X 0,Y 587.525,Z 530.163,A -85,B 0,C 180,E1 -1362.083,E2 -1362.083} C_VEL
LIN {X 0,Y 587.445,Z 540.778,A -85,B 0,C 180,E1 -1363.314,E2 -1363.314} C_VEL
LIN {X 0,Y 587.336,Z 551.157,A -85,B 0,C 180,E1 -1364.73,E2 -1364.73} C_VEL
LIN {X 0,Y 587.257,Z 559.882,A -85,B 0,C 180,E1 -1366.155,E2 -1366.155} C_VEL
LIN {X 0,Y 587.241,Z 566.34,A -85,B 0,C 180,E1 -1367.409,E2 -1367.409} C_VEL
LIN {X 0,Y 587.192,Z 573.098,A -85,B 0,C 180,E1 -1368.997,E2 -1368.997} C_VEL
LIN {X 0,Y 587.183,Z 577.506,A -85,B 0,C 180,E1 -1370.31,E2 -1370.31} C_VEL
LIN {X 0,Y 587.142,Z 581.328,A -85,B 0,C 180,E1 -1371.781,E2 -1371.781} C_VEL
LIN {X 0,Y 587.108,Z 584.034,A -85,B 0,C 180,E1 -1373.267,E2 -1373.267} C_VEL
LIN {X 0,Y 587.098,Z 585.544,A -85,B 0,C 180,E1 -1374.769,E2 -1374.769} C_VEL
LIN {X 0,Y 587.122,Z 585.951,A -85,B 0,C 180,E1 -1376.288,E2 -1376.288} C_VEL
LIN {X 0,Y 587.139,Z 585.193,A -85,B 0,C 180,E1 -1377.828,E2 -1377.828} C_VEL
LIN {X 0,Y 587.129,Z 583.121,A -85,B 0,C 180,E1 -1379.391,E2 -1379.391} C_VEL
LIN {X 0,Y 587.161,Z 579.735,A -85,B 0,C 180,E1 -1380.976,E2 -1380.976} C_VEL
LIN {X 0,Y 587.161,Z 574.903,A -85,B 0,C 180,E1 -1382.589,E2 -1382.589} C_VEL
LIN {X 0,Y 587.213,Z 570.207,A -85,B 0,C 180,E1 -1383.815,E2 -1383.815} C_VEL
LIN {X 0,Y 587.255,Z 563.306,A -85,B 0,C 180,E1 -1385.294,E2 -1385.294} C_VEL
LIN {X 0,Y 587.272,Z 555.062,A -85,B 0,C 180,E1 -1386.752,E2 -1386.752} C_VEL
LIN {X 0,Y 587.375,Z 545.754,A -85,B 0,C 180,E1 -1388.129,E2 -1388.129} C_VEL
LIN {X 0,Y 587.501,Z 534.171,A -85,B 0,C 180,E1 -1389.568,E2 -1389.568} C_VEL
LIN {X 0,Y 587.61,Z 522.537,A -85,B 0,C 180,E1 -1390.789,E2 -1390.789} C_VEL
LIN {X 0,Y 587.802,Z 509.927,A -85,B 0,C 180,E1 -1391.917,E2 -1391.917} C_VEL
LIN {X 0,Y 587.956,Z 496.43,A -85,B 0,C 180,E1 -1392.947,E2 -1392.947} C_VEL
LIN {X 0,Y 588.131,Z 482.046,A -85,B 0,C 180,E1 -1393.874,E2 -1393.874} C_VEL
LIN {X 0,Y 588.294,Z 467.924,A -85,B 0,C 180,E1 -1394.636,E2 -1394.636} C_VEL
LIN {X 0,Y 588.463,Z 452.739,A -85,B 0,C 180,E1 -1395.302,E2 -1395.302} C_VEL
LIN {X 0,Y 588.624,Z 436.658,A -85,B 0,C 180,E1 -1395.859,E2 -1395.859} C_VEL
LIN {X 0,Y 588.787,Z 419.698,A -85,B 0,C 180,E1 -1396.291,E2 -1396.291} C_VEL
LIN {X 0,Y 588.846,Z 402.682,A -85,B 0,C 180,E1 -1396.578,E2 -1396.578} C_VEL
LIN {X 0,Y 589.196,Z 210.972,A -85,B 0,C 180,E1 -1399.029,E2 -1399.029} C_VEL
LIN {X 0,Y 588.284,Z 205.712,A -85,B 0,C 180,E1 -1399.151,E2 -1399.151} C_VEL
LIN {X 0,Y 588.388,Z 189.314,A -85,B 0,C 180,E1 -1400.724,E2 -1400.724} C_VEL
LIN {X 0,Y 587.298,Z 184.645,A -85,B 0,C 180,E1 -1401.243,E2 -1401.243} C_VEL
LIN {X 0,Y 587.277,Z 184.64,A -85,B 0,C 180,E1 -1404.099,E2 -1404.099} C_VEL
LIN {X 0,Y 587.324,Z 184.638,A -85,B 0,C 180,E1 -1406.889,E2 -1406.889} C_VEL
LIN {X 0,Y 587.31,Z 184.639,A -85,B 0,C 180,E1 -1409.493,E2 -1409.493} C_VEL
LIN {X 0,Y 587.296,Z 184.637,A -85,B 0,C 180,E1 -1412.18,E2 -1412.18} C_VEL
LIN {X 0,Y 587.301,Z 184.638,A -85,B 0,C 180,E1 -1414.482,E2 -1414.482} C_VEL
LIN {X 0,Y 587.304,Z 184.641,A -85,B 0,C 180,E1 -1417.133,E2 -1417.133} C_VEL
LIN {X 0,Y 587.314,Z 184.634,A -85,B 0,C 180,E1 -1419.695,E2 -1419.695} C_VEL
LIN {X 0,Y 587.288,Z 184.637,A -85,B 0,C 180,E1 -1421.872,E2 -1421.872} C_VEL
LIN {X 0,Y 587.307,Z 184.635,A -85,B 0,C 180,E1 -1424.024,E2 -1424.024} C_VEL
LIN {X 0,Y 587.341,Z 184.633,A -85,B 0,C 180,E1 -1426.154,E2 -1426.154} C_VEL
LIN {X 0,Y 587.334,Z 184.635,A -85,B 0,C 180,E1 -1428.962,E2 -1428.962} C_VEL
LIN {X 0,Y 587.33,Z 184.632,A -85,B 0,C 180,E1 -1431.744,E2 -1431.744} C_VEL
LIN {X 0,Y 587.351,Z 184.638,A -85,B 0,C 180,E1 -1434.507,E2 -1434.507} C_VEL
LIN {X 0,Y 587.363,Z 184.628,A -85,B 0,C 180,E1 -1437.257,E2 -1437.257} C_VEL
LIN {X 0,Y 587.371,Z 184.632,A -85,B 0,C 180,E1 -1440,E2 -1440} C_VEL
LIN {X 0,Y 587.372,Z 184.629,A -85,B 0,C 180,E1 -1442.743,E2 -1442.743} C_VEL
LIN {X 0,Y 587.346,Z 184.631,A -85,B 0,C 180,E1 -1445.493,E2 -1445.493} C_VEL
LIN {X 0,Y 587.364,Z 184.635,A -85,B 0,C 180,E1 -1448.255,E2 -1448.255} C_VEL
LIN {X 0,Y 587.34,Z 184.63,A -85,B 0,C 180,E1 -1451.134,E2 -1451.134} C_VEL
LIN {X 0,Y 587.359,Z 184.633,A -85,B 0,C 180,E1 -1454.261,E2 -1454.261} C_VEL
LIN {X 0,Y 587.353,Z 184.632,A -85,B 0,C 180,E1 -1457.406,E2 -1457.406} C_VEL
LIN {X 0,Y 587.325,Z 184.635,A -85,B 0,C 180,E1 -1460.305,E2 -1460.305} C_VEL
LIN {X 0,Y 587.318,Z 184.636,A -85,B 0,C 180,E1 -1463.259,E2 -1463.259} C_VEL
LIN {X 0,Y 587.334,Z 184.639,A -85,B 0,C 180,E1 -1465.517,E2 -1465.517} C_VEL
LIN {X 0,Y 587.343,Z 184.636,A -85,B 0,C 180,E1 -1467.818,E2 -1467.818} C_VEL
LIN {X 0,Y 587.335,Z 184.631,A -85,B 0,C 180,E1 -1470.511,E2 -1470.511} C_VEL
LIN {X 0,Y 587.335,Z 184.636,A -85,B 0,C 180,E1 -1473.113,E2 -1473.113} C_VEL
LIN {X 0,Y 587.296,Z 184.644,A -85,B 0,C 180,E1 -1475.539,E2 -1475.539} C_VEL
LIN {X 0,Y 587.332,Z 184.635,A -85,B 0,C 180,E1 -1477.839,E2 -1477.839} C_VEL
LIN {X 0,Y 587.312,Z 184.634,A -85,B 0,C 180,E1 -1480.254,E2 -1480.254} C_VEL
LIN {X 0,Y 587.312,Z 184.644,A -85,B 0,C 180,E1 -1483.119,E2 -1483.119} C_VEL
LIN {X 0,Y 587.306,Z 184.635,A -85,B 0,C 180,E1 -1486.049,E2 -1486.049} C_VEL
LIN {X 0,Y 587.332,Z 184.64,A -85,B 0,C 180,E1 -1488.925,E2 -1488.925} C_VEL
LIN {X 0,Y 587.319,Z 184.636,A -85,B 0,C 180,E1 -1491.521,E2 -1491.521} C_VEL
LIN {X 0,Y 587.285,Z 184.638,A -85,B 0,C 180,E1 -1494.1,E2 -1494.1} C_VEL
LIN {X 0,Y 587.328,Z 184.638,A -85,B 0,C 180,E1 -1496.604,E2 -1496.604} C_VEL
LIN {X 0,Y 587.329,Z 184.64,A -85,B 0,C 180,E1 -1499.034,E2 -1499.034} C_VEL
LIN {X 0,Y 587.305,Z 184.639,A -85,B 0,C 180,E1 -1501.403,E2 -1501.403} C_VEL
LIN {X 0,Y 587.358,Z 184.819,A -85,B 0,C 180,E1 -1502.55,E2 -1502.55} C_VEL
LIN {X 0,Y 588.675,Z 189.472,A -85,B 0,C 180,E1 -1503.021,E2 -1503.021} C_VEL
LIN {X 0,Y 588.837,Z 197.054,A -85,B 0,C 180,E1 -1503.686,E2 -1503.686} C_VEL
LIN {X 0,Y 588.504,Z 230.325,A -85,B 0,C 180,E1 -1506.512,E2 -1506.512} C_VEL
LIN {X 0,Y 588.488,Z 234.982,A -85,B 0,C 180,E1 -1506.904,E2 -1506.904} C_VEL
LIN {X 0,Y 589.247,Z 240.685,A -85,B 0,C 180,E1 -1507.014,E2 -1507.014} C_VEL
LIN {X 0,Y 588.774,Z 442.457,A -85,B 0,C 180,E1 -1509.611,E2 -1509.611} C_VEL
LIN {X 0,Y 588.703,Z 459.021,A -85,B 0,C 180,E1 -1509.973,E2 -1509.973} C_VEL
LIN {X 0,Y 588.552,Z 475.252,A -85,B 0,C 180,E1 -1510.467,E2 -1510.467} C_VEL
LIN {X 0,Y 588.342,Z 491.979,A -85,B 0,C 180,E1 -1511.134,E2 -1511.134} C_VEL
LIN {X 0,Y 588.2,Z 507.313,A -85,B 0,C 180,E1 -1511.902,E2 -1511.902} C_VEL
LIN {X 0,Y 588.036,Z 521.566,A -85,B 0,C 180,E1 -1512.762,E2 -1512.762} C_VEL
LIN {X 0,Y 587.857,Z 535.544,A -85,B 0,C 180,E1 -1513.773,E2 -1513.773} C_VEL
LIN {X 0,Y 587.676,Z 547.076,A -85,B 0,C 180,E1 -1514.747,E2 -1514.747} C_VEL
LIN {X 0,Y 587.578,Z 559.627,A -85,B 0,C 180,E1 -1515.982,E2 -1515.982} C_VEL
LIN {X 0,Y 587.426,Z 570.336,A -85,B 0,C 180,E1 -1517.213,E2 -1517.213} C_VEL
LIN {X 0,Y 587.351,Z 580.679,A -85,B 0,C 180,E1 -1518.614,E2 -1518.614} C_VEL
LIN {X 0,Y 587.29,Z 589.288,A -85,B 0,C 180,E1 -1520.008,E2 -1520.008} C_VEL
LIN {X 0,Y 587.239,Z 596.489,A -85,B 0,C 180,E1 -1521.397,E2 -1521.397} C_VEL
LIN {X 0,Y 587.207,Z 602.469,A -85,B 0,C 180,E1 -1522.781,E2 -1522.781} C_VEL
LIN {X 0,Y 587.188,Z 608.247,A -85,B 0,C 180,E1 -1524.506,E2 -1524.506} C_VEL
LIN {X 0,Y 587.167,Z 611.635,A -85,B 0,C 180,E1 -1525.882,E2 -1525.882} C_VEL
LIN {X 0,Y 587.119,Z 614.088,A -85,B 0,C 180,E1 -1527.256,E2 -1527.256} C_VEL
LIN {X 0,Y 587.14,Z 615.479,A -85,B 0,C 180,E1 -1528.628,E2 -1528.628} C_VEL
LIN {X 0,Y 587.132,Z 616,A -85,B 0,C 180,E1 -1530,E2 -1530} C_VEL
LIN {X 0,Y 587.14,Z 615.478,A -85,B 0,C 180,E1 -1531.372,E2 -1531.372} C_VEL
LIN {X 0,Y 587.119,Z 614.087,A -85,B 0,C 180,E1 -1532.745,E2 -1532.745} C_VEL
LIN {X 0,Y 587.167,Z 611.634,A -85,B 0,C 180,E1 -1534.118,E2 -1534.118} C_VEL
LIN {X 0,Y 587.188,Z 607.186,A -85,B 0,C 180,E1 -1535.839,E2 -1535.839} C_VEL
LIN {X 0,Y 587.208,Z 602.468,A -85,B 0,C 180,E1 -1537.22,E2 -1537.22} C_VEL
LIN {X 0,Y 587.245,Z 594.857,A -85,B 0,C 180,E1 -1538.951,E2 -1538.951} C_VEL
LIN {X 0,Y 587.302,Z 586.248,A -85,B 0,C 180,E1 -1540.515,E2 -1540.515} C_VEL
LIN {X 0,Y 587.366,Z 576.971,A -85,B 0,C 180,E1 -1541.912,E2 -1541.912} C_VEL
LIN {X 0,Y 587.449,Z 567.424,A -85,B 0,C 180,E1 -1543.139,E2 -1543.139} C_VEL
LIN {X 0,Y 587.589,Z 555.57,A -85,B 0,C 180,E1 -1544.441,E2 -1544.441} C_VEL
LIN {X 0,Y 587.759,Z 543.096,A -85,B 0,C 180,E1 -1545.607,E2 -1545.607} C_VEL
LIN {X 0,Y 587.909,Z 529.706,A -85,B 0,C 180,E1 -1546.673,E2 -1546.673} C_VEL
LIN {X 0,Y 588.087,Z 515.007,A -85,B 0,C 180,E1 -1547.653,E2 -1547.653} C_VEL
LIN {X 0,Y 588.288,Z 500.523,A -85,B 0,C 180,E1 -1548.456,E2 -1548.456} C_VEL
LIN {X 0,Y 588.444,Z 485.395,A -85,B 0,C 180,E1 -1549.149,E2 -1549.149} C_VEL
LIN {X 0,Y 588.617,Z 469.251,A -85,B 0,C 180,E1 -1549.735,E2 -1549.735} C_VEL
LIN {X 0,Y 588.746,Z 452.605,A -85,B 0,C 180,E1 -1550.185,E2 -1550.185} C_VEL
LIN {X 0,Y 588.812,Z 436.425,A -85,B 0,C 180,E1 -1550.479,E2 -1550.479} C_VEL
LIN {X 0,Y 589.25,Z 239.678,A -85,B 0,C 180,E1 -1552.999,E2 -1552.999} C_VEL
LIN {X 0,Y 588.479,Z 235.007,A -85,B 0,C 180,E1 -1553.094,E2 -1553.094} C_VEL
LIN {X 0,Y 588.836,Z 200.508,A -85,B 0,C 180,E1 -1556.016,E2 -1556.016} C_VEL
LIN {X 0,Y 588.673,Z 189.467,A -85,B 0,C 180,E1 -1556.979,E2 -1556.979} C_VEL
LIN {X 0,Y 587.351,Z 184.64,A -85,B 0,C 180,E1 -1557.475,E2 -1557.475} C_VEL
LIN {X 0,Y 587.311,Z 184.635,A -85,B 0,C 180,E1 -1560.171,E2 -1560.171} C_VEL
LIN {X 0,Y 587.325,Z 184.633,A -85,B 0,C 180,E1 -1562.58,E2 -1562.58} C_VEL
LIN {X 0,Y 587.318,Z 184.642,A -85,B 0,C 180,E1 -1565.056,E2 -1565.056} C_VEL
LIN {X 0,Y 587.328,Z 184.633,A -85,B 0,C 180,E1 -1567.837,E2 -1567.837} C_VEL
LIN {X 0,Y 587.307,Z 184.634,A -85,B 0,C 180,E1 -1570.255,E2 -1570.255} C_VEL
LIN {X 0,Y 587.3,Z 184.645,A -85,B 0,C 180,E1 -1573.117,E2 -1573.117} C_VEL
LIN {X 0,Y 587.294,Z 184.635,A -85,B 0,C 180,E1 -1576.047,E2 -1576.047} C_VEL
LIN {X 0,Y 587.33,Z 184.641,A -85,B 0,C 180,E1 -1578.925,E2 -1578.925} C_VEL
LIN {X 0,Y 587.317,Z 184.635,A -85,B 0,C 180,E1 -1581.52,E2 -1581.52} C_VEL
LIN {X 0,Y 587.285,Z 184.636,A -85,B 0,C 180,E1 -1584.1,E2 -1584.1} C_VEL
LIN {X 0,Y 587.333,Z 184.639,A -85,B 0,C 180,E1 -1586.889,E2 -1586.889} C_VEL
LIN {X 0,Y 587.324,Z 184.633,A -85,B 0,C 180,E1 -1589.491,E2 -1589.491} C_VEL
LIN {X 0,Y 587.347,Z 184.633,A -85,B 0,C 180,E1 -1592.307,E2 -1592.307} C_VEL
LIN {X 0,Y 587.345,Z 184.631,A -85,B 0,C 180,E1 -1595.241,E2 -1595.241} C_VEL
LIN {X 0,Y 587.313,Z 184.637,A -85,B 0,C 180,E1 -1598.225,E2 -1598.225} C_VEL
LIN {X 0,Y 587.343,Z 184.63,A -85,B 0,C 180,E1 -1601.151,E2 -1601.151} C_VEL
LIN {X 0,Y 587.314,Z 184.636,A -85,B 0,C 180,E1 -1604.025,E2 -1604.025} C_VEL
LIN {X 0,Y 587.346,Z 184.634,A -85,B 0,C 180,E1 -1606.154,E2 -1606.154} C_VEL
LIN {X 0,Y 587.337,Z 184.631,A -85,B 0,C 180,E1 -1608.962,E2 -1608.962} C_VEL
LIN {X 0,Y 587.335,Z 184.632,A -85,B 0,C 180,E1 -1611.744,E2 -1611.744} C_VEL
LIN {X 0,Y 587.354,Z 184.635,A -85,B 0,C 180,E1 -1614.507,E2 -1614.507} C_VEL
LIN {X 0,Y 587.365,Z 184.623,A -85,B 0,C 180,E1 -1617.257,E2 -1617.257} C_VEL
LIN {X 0,Y 587.375,Z 184.63,A -85,B 0,C 180,E1 -1620,E2 -1620} C_VEL
LIN {X 0,Y 587.373,Z 184.628,A -85,B 0,C 180,E1 -1622.743,E2 -1622.743} C_VEL
LIN {X 0,Y 587.348,Z 184.628,A -85,B 0,C 180,E1 -1625.493,E2 -1625.493} C_VEL
LIN {X 0,Y 587.361,Z 184.636,A -85,B 0,C 180,E1 -1628.255,E2 -1628.255} C_VEL
LIN {X 0,Y 587.344,Z 184.628,A -85,B 0,C 180,E1 -1631.134,E2 -1631.134} C_VEL
LIN {X 0,Y 587.361,Z 184.634,A -85,B 0,C 180,E1 -1634.261,E2 -1634.261} C_VEL
LIN {X 0,Y 587.353,Z 184.63,A -85,B 0,C 180,E1 -1637.406,E2 -1637.406} C_VEL
LIN {X 0,Y 587.321,Z 184.635,A -85,B 0,C 180,E1 -1638.317,E2 -1638.317} C_VEL
LIN {X 0,Y 586.668,Z 184.714,A -85,B 0,C 180,E1 -1638.889,E2 -1638.889} C_VEL
LIN {X 0,Y 583.835,Z 185.073,A -85,B 0,C 180,E1 -1639.817,E2 -1639.817} C_VEL
LIN {X 0,Y 581.425,Z 185.371,A -85,B 0,C 180,E1 -1640.564,E2 -1640.564} C_VEL
LIN {X 0,Y 580.374,Z 185.499,A -85,B 0,C 180,E1 -1641.14,E2 -1641.14} C_VEL
LIN {X 0,Y 580.279,Z 185.511,A -85,B 0,C 180,E1 -1641.336,E2 -1641.336} C_VEL
LIN {X 0,Y 580.298,Z 185.509,A -85,B 0,C 180,E1 -1644.316,E2 -1644.316} C_VEL
LIN {X 0,Y 580.274,Z 185.51,A -85,B 0,C 180,E1 -1646.623,E2 -1646.623} C_VEL
LIN {X 0,Y 580.303,Z 185.51,A -85,B 0,C 180,E1 -1649.311,E2 -1649.311} C_VEL
LIN {X 0,Y 580.296,Z 185.509,A -85,B 0,C 180,E1 -1652.201,E2 -1652.201} C_VEL
LIN {X 0,Y 580.298,Z 185.507,A -85,B 0,C 180,E1 -1654.696,E2 -1654.696} C_VEL
LIN {X 0,Y 580.296,Z 185.511,A -85,B 0,C 180,E1 -1657.268,E2 -1657.268} C_VEL
LIN {X 0,Y 580.29,Z 185.51,A -85,B 0,C 180,E1 -1660.271,E2 -1660.271} C_VEL
LIN {X 0,Y 580.275,Z 185.51,A -85,B 0,C 180,E1 -1662.706,E2 -1662.706} C_VEL
LIN {X 0,Y 580.267,Z 185.52,A -85,B 0,C 180,E1 -1665.609,E2 -1665.609} C_VEL
LIN {X 0,Y 580.287,Z 185.508,A -85,B 0,C 180,E1 -1668.232,E2 -1668.232} C_VEL
LIN {X 0,Y 580.276,Z 185.513,A -85,B 0,C 180,E1 -1670.965,E2 -1670.965} C_VEL
LIN {X 0,Y 580.267,Z 185.516,A -85,B 0,C 180,E1 -1673.597,E2 -1673.597} C_VEL
LIN {X 0,Y 580.318,Z 185.506,A -85,B 0,C 180,E1 -1676.146,E2 -1676.146} C_VEL
LIN {X 0,Y 580.28,Z 185.51,A -85,B 0,C 180,E1 -1678.615,E2 -1678.615} C_VEL
LIN {X 0,Y 580.292,Z 185.515,A -85,B 0,C 180,E1 -1681.024,E2 -1681.024} C_VEL
LIN {X 0,Y 580.292,Z 185.511,A -85,B 0,C 180,E1 -1683.666,E2 -1683.666} C_VEL
LIN {X 0,Y 580.299,Z 185.509,A -85,B 0,C 180,E1 -1685.684,E2 -1685.684} C_VEL
LIN {X 0,Y 580.269,Z 185.512,A -85,B 0,C 180,E1 -1687.947,E2 -1687.947} C_VEL
LIN {X 0,Y 580.296,Z 185.513,A -85,B 0,C 180,E1 -1690.913,E2 -1690.913} C_VEL
LIN {X 0,Y 580.267,Z 185.512,A -85,B 0,C 180,E1 -1693.825,E2 -1693.825} C_VEL
LIN {X 0,Y 580.327,Z 185.501,A -85,B 0,C 180,E1 -1695.983,E2 -1695.983} C_VEL
LIN {X 0,Y 580.305,Z 185.515,A -85,B 0,C 180,E1 -1698.827,E2 -1698.827} C_VEL
LIN {X 0,Y 580.326,Z 185.505,A -85,B 0,C 180,E1 -1701.644,E2 -1701.644} C_VEL
LIN {X 0,Y 580.331,Z 185.506,A -85,B 0,C 180,E1 -1704.44,E2 -1704.44} C_VEL
LIN {X 0,Y 580.331,Z 185.509,A -85,B 0,C 180,E1 -1707.223,E2 -1707.223} C_VEL
LIN {X 0,Y 580.352,Z 185.508,A -85,B 0,C 180,E1 -1710.347,E2 -1710.347} C_VEL
LIN {X 0,Y 580.388,Z 185.741,A -85,B 0,C 180,E1 -1710.65,E2 -1710.65} C_VEL
LIN {X 0,Y 581.605,Z 190.873,A -85,B 0,C 180,E1 -1711.211,E2 -1711.211} C_VEL
LIN {X 0,Y 581.548,Z 205.776,A -85,B 0,C 180,E1 -1712.662,E2 -1712.662} C_VEL
LIN {X 0,Y 582.717,Z 212.356,A -85,B 0,C 180,E1 -1712.808,E2 -1712.808} C_VEL
LIN {X 0,Y 582.188,Z 410.803,A -85,B 0,C 180,E1 -1715.39,E2 -1715.39} C_VEL
LIN {X 0,Y 582.041,Z 427.499,A -85,B 0,C 180,E1 -1715.739,E2 -1715.739} C_VEL
LIN {X 0,Y 581.842,Z 443.032,A -85,B 0,C 180,E1 -1716.197,E2 -1716.197} C_VEL
LIN {X 0,Y 581.688,Z 458.828,A -85,B 0,C 180,E1 -1716.808,E2 -1716.808} C_VEL
LIN {X 0,Y 581.425,Z 474.293,A -85,B 0,C 180,E1 -1717.561,E2 -1717.561} C_VEL
LIN {X 0,Y 581.208,Z 488.965,A -85,B 0,C 180,E1 -1718.431,E2 -1718.431} C_VEL
LIN {X 0,Y 580.978,Z 502.694,A -85,B 0,C 180,E1 -1719.399,E2 -1719.399} C_VEL
LIN {X 0,Y 580.788,Z 515.477,A -85,B 0,C 180,E1 -1720.457,E2 -1720.457} C_VEL
LIN {X 0,Y 580.582,Z 528.29,A -85,B 0,C 180,E1 -1721.706,E2 -1721.706} C_VEL
LIN {X 0,Y 580.442,Z 539.073,A -85,B 0,C 180,E1 -1722.944,E2 -1722.944} C_VEL
LIN {X 0,Y 580.315,Z 549.43,A -85,B 0,C 180,E1 -1724.339,E2 -1724.339} C_VEL
LIN {X 0,Y 580.206,Z 558.639,A -85,B 0,C 180,E1 -1725.815,E2 -1725.815} C_VEL
LIN {X 0,Y 580.172,Z 566.163,A -85,B 0,C 180,E1 -1727.264,E2 -1727.264} C_VEL
LIN {X 0,Y 580.126,Z 572.419,A -85,B 0,C 180,E1 -1728.725,E2 -1728.725} C_VEL
LIN {X 0,Y 580.086,Z 577.385,A -85,B 0,C 180,E1 -1730.199,E2 -1730.199} C_VEL
LIN {X 0,Y 580.047,Z 580.399,A -85,B 0,C 180,E1 -1731.314,E2 -1731.314} C_VEL
LIN {X 0,Y 580.042,Z 583.585,A -85,B 0,C 180,E1 -1732.951,E2 -1732.951} C_VEL
LIN {X 0,Y 580.003,Z 585.482,A -85,B 0,C 180,E1 -1734.662,E2 -1734.662} C_VEL
LIN {X 0,Y 580.042,Z 585.952,A -85,B 0,C 180,E1 -1736.284,E2 -1736.284} C_VEL
LIN {X 0,Y 580.04,Z 585.222,A -85,B 0,C 180,E1 -1737.811,E2 -1737.811} C_VEL
LIN {X 0,Y 580.065,Z 583.381,A -85,B 0,C 180,E1 -1739.268,E2 -1739.268} C_VEL
LIN {X 0,Y 580.066,Z 580.696,A -85,B 0,C 180,E1 -1740.658,E2 -1740.658} C_VEL
LIN {X 0,Y 580.08,Z 576.403,A -85,B 0,C 180,E1 -1742.213,E2 -1742.213} C_VEL
LIN {X 0,Y 580.12,Z 571.681,A -85,B 0,C 180,E1 -1743.548,E2 -1743.548} C_VEL
LIN {X 0,Y 580.164,Z 564.741,A -85,B 0,C 180,E1 -1745.127,E2 -1745.127} C_VEL
LIN {X 0,Y 580.204,Z 556.394,A -85,B 0,C 180,E1 -1746.666,E2 -1746.666} C_VEL
LIN {X 0,Y 580.346,Z 546.713,A -85,B 0,C 180,E1 -1748.141,E2 -1748.141} C_VEL
LIN {X 0,Y 580.469,Z 535.911,A -85,B 0,C 180,E1 -1749.527,E2 -1749.527} C_VEL
LIN {X 0,Y 580.613,Z 524.071,A -85,B 0,C 180,E1 -1750.816,E2 -1750.816} C_VEL
LIN {X 0,Y 580.827,Z 511.809,A -85,B 0,C 180,E1 -1751.952,E2 -1751.952} C_VEL
LIN {X 0,Y 581.058,Z 498.748,A -85,B 0,C 180,E1 -1752.989,E2 -1752.989} C_VEL
LIN {X 0,Y 581.285,Z 484.862,A -85,B 0,C 180,E1 -1753.922,E2 -1753.922} C_VEL
LIN {X 0,Y 581.523,Z 470.11,A -85,B 0,C 180,E1 -1754.746,E2 -1754.746} C_VEL
LIN {X 0,Y 581.714,Z 454.472,A -85,B 0,C 180,E1 -1755.463,E2 -1755.463} C_VEL
LIN {X 0,Y 581.912,Z 437.843,A -85,B 0,C 180,E1 -1756.06,E2 -1756.06} C_VEL
LIN {X 0,Y 582.082,Z 421.303,A -85,B 0,C 180,E1 -1756.499,E2 -1756.499} C_VEL
LIN {X 0,Y 582.197,Z 404.098,A -85,B 0,C 180,E1 -1756.804,E2 -1756.804} C_VEL
LIN {X 0,Y 582.694,Z 212.933,A -85,B 0,C 180,E1 -1759.275,E2 -1759.275} C_VEL
LIN {X 0,Y 581.879,Z 207.704,A -85,B 0,C 180,E1 -1759.378,E2 -1759.378} C_VEL
LIN {X 0,Y 581.496,Z 205.74,A -85,B 0,C 180,E1 -1759.433,E2 -1759.433} C_VEL
LIN {X 0,Y 581.667,Z 191.645,A -85,B 0,C 180,E1 -1760.8,E2 -1760.8} C_VEL
LIN {X 0,Y 580.263,Z 185.521,A -85,B 0,C 180,E1 -1761.493,E2 -1761.493} C_VEL
LIN {X 0,Y 580.233,Z 185.518,A -85,B 0,C 180,E1 -1764.244,E2 -1764.244} C_VEL
LIN {X 0,Y 580.276,Z 185.518,A -85,B 0,C 180,E1 -1766.974,E2 -1766.974} C_VEL
LIN {X 0,Y 580.271,Z 185.517,A -85,B 0,C 180,E1 -1769.424,E2 -1769.424} C_VEL
LIN {X 0,Y 580.25,Z 185.515,A -85,B 0,C 180,E1 -1772.149,E2 -1772.149} C_VEL
LIN {X 0,Y 580.27,Z 185.52,A -85,B 0,C 180,E1 -1774.919,E2 -1774.919} C_VEL
LIN {X 0,Y 580.247,Z 185.513,A -85,B 0,C 180,E1 -1777.946,E2 -1777.946} C_VEL
LIN {X 0,Y 580.291,Z 185.517,A -85,B 0,C 180,E1 -1780.913,E2 -1780.913} C_VEL
LIN {X 0,Y 580.263,Z 185.512,A -85,B 0,C 180,E1 -1783.825,E2 -1783.825} C_VEL
LIN {X 0,Y 580.309,Z 185.507,A -85,B 0,C 180,E1 -1785.983,E2 -1785.983} C_VEL
LIN {X 0,Y 580.297,Z 185.514,A -85,B 0,C 180,E1 -1788.827,E2 -1788.827} C_VEL
LIN {X 0,Y 580.3,Z 185.507,A -85,B 0,C 180,E1 -1791.644,E2 -1791.644} C_VEL
LIN {X 0,Y 580.316,Z 185.515,A -85,B 0,C 180,E1 -1794.44,E2 -1794.44} C_VEL
LIN {X 0,Y 580.33,Z 185.504,A -85,B 0,C 180,E1 -1797.223,E2 -1797.223} C_VEL
LIN {X 0,Y 580.341,Z 185.507,A -85,B 0,C 180,E1 -1800,E2 -1800} C_VEL
LIN {X 0,Y 580.337,Z 185.505,A -85,B 0,C 180,E1 -1802.777,E2 -1802.777} C_VEL
LIN {X 0,Y 580.313,Z 185.507,A -85,B 0,C 180,E1 -1805.56,E2 -1805.56} C_VEL
LIN {X 0,Y 580.328,Z 185.51,A -85,B 0,C 180,E1 -1808.356,E2 -1808.356} C_VEL
LIN {X 0,Y 580.292,Z 185.508,A -85,B 0,C 180,E1 -1811.191,E2 -1811.191} C_VEL
LIN {X 0,Y 580.32,Z 185.514,A -85,B 0,C 180,E1 -1814.017,E2 -1814.017} C_VEL
LIN {X 0,Y 580.305,Z 185.506,A -85,B 0,C 180,E1 -1816.914,E2 -1816.914} C_VEL
LIN {X 0,Y 580.299,Z 185.517,A -85,B 0,C 180,E1 -1819.822,E2 -1819.822} C_VEL
LIN {X 0,Y 580.29,Z 185.509,A -85,B 0,C 180,E1 -1822.803,E2 -1822.803} C_VEL
LIN {X 0,Y 580.303,Z 185.509,A -85,B 0,C 180,E1 -1825.08,E2 -1825.08} C_VEL
LIN {X 0,Y 580.314,Z 185.511,A -85,B 0,C 180,E1 -1827.863,E2 -1827.863} C_VEL
LIN {X 0,Y 580.286,Z 185.51,A -85,B 0,C 180,E1 -1830.696,E2 -1830.696} C_VEL
LIN {X 0,Y 580.299,Z 185.516,A -85,B 0,C 180,E1 -1833.317,E2 -1833.317} C_VEL
LIN {X 0,Y 580.243,Z 185.519,A -85,B 0,C 180,E1 -1835.757,E2 -1835.757} C_VEL
LIN {X 0,Y 580.281,Z 185.511,A -85,B 0,C 180,E1 -1838.147,E2 -1838.147} C_VEL
LIN {X 0,Y 580.294,Z 185.512,A -85,B 0,C 180,E1 -1840.844,E2 -1840.844} C_VEL
LIN {X 0,Y 580.273,Z 185.515,A -85,B 0,C 180,E1 -1843.658,E2 -1843.658} C_VEL
LIN {X 0,Y 580.269,Z 185.515,A -85,B 0,C 180,E1 -1846.61,E2 -1846.61} C_VEL
LIN {X 0,Y 580.294,Z 185.517,A -85,B 0,C 180,E1 -1849.157,E2 -1849.157} C_VEL
LIN {X 0,Y 580.282,Z 185.51,A -85,B 0,C 180,E1 -1851.928,E2 -1851.928} C_VEL
LIN {X 0,Y 580.247,Z 185.518,A -85,B 0,C 180,E1 -1854.453,E2 -1854.453} C_VEL
LIN {X 0,Y 580.283,Z 185.518,A -85,B 0,C 180,E1 -1856.975,E2 -1856.975} C_VEL
LIN {X 0,Y 580.284,Z 185.513,A -85,B 0,C 180,E1 -1859.425,E2 -1859.425} C_VEL
LIN {X 0,Y 580.298,Z 185.518,A -85,B 0,C 180,E1 -1862.26,E2 -1862.26} C_VEL
LIN {X 0,Y 582.183,Z 192.683,A -85,B 0,C 180,E1 -1862.978,E2 -1862.978} C_VEL
LIN {X 0,Y 581.927,Z 220.416,A -85,B 0,C 180,E1 -1865.379,E2 -1865.379} C_VEL
LIN {X 0,Y 581.768,Z 234.896,A -85,B 0,C 180,E1 -1866.614,E2 -1866.614} C_VEL
LIN {X 0,Y 582.717,Z 241.175,A -85,B 0,C 180,E1 -1866.748,E2 -1866.748} C_VEL
LIN {X 0,Y 582.124,Z 442.457,A -85,B 0,C 180,E1 -1869.367,E2 -1869.367} C_VEL
LIN {X 0,Y 582.036,Z 459.023,A -85,B 0,C 180,E1 -1869.733,E2 -1869.733} C_VEL
LIN {X 0,Y 581.831,Z 475.255,A -85,B 0,C 180,E1 -1870.232,E2 -1870.232} C_VEL
LIN {X 0,Y 581.599,Z 492.058,A -85,B 0,C 180,E1 -1870.91,E2 -1870.91} C_VEL
LIN {X 0,Y 581.414,Z 507.31,A -85,B 0,C 180,E1 -1871.683,E2 -1871.683} C_VEL
LIN {X 0,Y 581.161,Z 521.788,A -85,B 0,C 180,E1 -1872.567,E2 -1872.567} C_VEL
LIN {X 0,Y 580.977,Z 535.547,A -85,B 0,C 180,E1 -1873.575,E2 -1873.575} C_VEL
LIN {X 0,Y 580.742,Z 547.076,A -85,B 0,C 180,E1 -1874.56,E2 -1874.56} C_VEL
LIN {X 0,Y 580.589,Z 558.624,A -85,B 0,C 180,E1 -1875.7,E2 -1875.7} C_VEL
LIN {X 0,Y 580.412,Z 570.338,A -85,B 0,C 180,E1 -1877.056,E2 -1877.056} C_VEL
LIN {X 0,Y 580.315,Z 580.678,A -85,B 0,C 180,E1 -1878.474,E2 -1878.474} C_VEL
LIN {X 0,Y 580.219,Z 589.287,A -85,B 0,C 180,E1 -1879.885,E2 -1879.885} C_VEL
LIN {X 0,Y 580.164,Z 596.49,A -85,B 0,C 180,E1 -1881.291,E2 -1881.291} C_VEL
LIN {X 0,Y 580.119,Z 602.468,A -85,B 0,C 180,E1 -1882.692,E2 -1882.692} C_VEL
LIN {X 0,Y 580.112,Z 608.248,A -85,B 0,C 180,E1 -1884.438,E2 -1884.438} C_VEL
LIN {X 0,Y 580.085,Z 611.636,A -85,B 0,C 180,E1 -1885.832,E2 -1885.832} C_VEL
LIN {X 0,Y 580.031,Z 614.089,A -85,B 0,C 180,E1 -1887.222,E2 -1887.222} C_VEL
LIN {X 0,Y 580.04,Z 615.479,A -85,B 0,C 180,E1 -1888.612,E2 -1888.612} C_VEL
LIN {X 0,Y 580.033,Z 616,A -85,B 0,C 180,E1 -1890,E2 -1890} C_VEL
LIN {X 0,Y 580.04,Z 615.479,A -85,B 0,C 180,E1 -1891.389,E2 -1891.389} C_VEL
LIN {X 0,Y 580.031,Z 614.087,A -85,B 0,C 180,E1 -1892.778,E2 -1892.778} C_VEL
LIN {X 0,Y 580.085,Z 611.635,A -85,B 0,C 180,E1 -1894.169,E2 -1894.169} C_VEL
LIN {X 0,Y 580.099,Z 607.187,A -85,B 0,C 180,E1 -1895.911,E2 -1895.911} C_VEL
LIN {X 0,Y 580.119,Z 602.468,A -85,B 0,C 180,E1 -1897.308,E2 -1897.308} C_VEL
LIN {X 0,Y 580.157,Z 594.857,A -85,B 0,C 180,E1 -1899.061,E2 -1899.061} C_VEL
LIN {X 0,Y 580.24,Z 586.249,A -85,B 0,C 180,E1 -1900.644,E2 -1900.644} C_VEL
LIN {X 0,Y 580.335,Z 576.972,A -85,B 0,C 180,E1 -1902.058,E2 -1902.058} C_VEL
LIN {X 0,Y 580.44,Z 567.423,A -85,B 0,C 180,E1 -1903.3,E2 -1903.3} C_VEL
LIN {X 0,Y 580.623,Z 555.931,A -85,B 0,C 180,E1 -1904.582,E2 -1904.582} C_VEL
LIN {X 0,Y 580.814,Z 544.142,A -85,B 0,C 180,E1 -1905.708,E2 -1905.708} C_VEL
LIN {X 0,Y 581.011,Z 530.876,A -85,B 0,C 180,E1 -1906.786,E2 -1906.786} C_VEL
LIN {X 0,Y 581.235,Z 516.43,A -85,B 0,C 180,E1 -1907.777,E2 -1907.777} C_VEL
LIN {X 0,Y 581.479,Z 502.274,A -85,B 0,C 180,E1 -1908.589,E2 -1908.589} C_VEL
LIN {X 0,Y 581.697,Z 487.012,A -85,B 0,C 180,E1 -1909.314,E2 -1909.314} C_VEL
LIN {X 0,Y 581.902,Z 471.345,A -85,B 0,C 180,E1 -1909.903,E2 -1909.903} C_VEL
LIN {X 0,Y 582.043,Z 455.353,A -85,B 0,C 180,E1 -1910.359,E2 -1910.359} C_VEL
LIN {X 0,Y 582.144,Z 439.437,A -85,B 0,C 180,E1 -1910.678,E2 -1910.678} C_VEL
LIN {X 0,Y 582.718,Z 240.338,A -85,B 0,C 180,E1 -1913.263,E2 -1913.263} C_VEL
LIN {X 0,Y 581.754,Z 234.947,A -85,B 0,C 180,E1 -1913.382,E2 -1913.382} C_VEL
LIN {X 0,Y 582.175,Z 201.612,A -85,B 0,C 180,E1 -1916.24,E2 -1916.24} C_VEL
LIN {X 0,Y 582.176,Z 192.675,A -85,B 0,C 180,E1 -1917.023,E2 -1917.023} C_VEL
LIN {X 0,Y 580.3,Z 185.515,A -85,B 0,C 180,E1 -1917.765,E2 -1917.765} C_VEL
LIN {X 0,Y 580.267,Z 185.515,A -85,B 0,C 180,E1 -1920.692,E2 -1920.692} C_VEL
LIN {X 0,Y 580.298,Z 185.515,A -85,B 0,C 180,E1 -1923.316,E2 -1923.316} C_VEL
LIN {X 0,Y 580.24,Z 185.518,A -85,B 0,C 180,E1 -1925.756,E2 -1925.756} C_VEL
LIN {X 0,Y 580.28,Z 185.51,A -85,B 0,C 180,E1 -1928.147,E2 -1928.147} C_VEL
LIN {X 0,Y 580.294,Z 185.513,A -85,B 0,C 180,E1 -1930.843,E2 -1930.843} C_VEL
LIN {X 0,Y 580.266,Z 185.513,A -85,B 0,C 180,E1 -1933.659,E2 -1933.659} C_VEL
LIN {X 0,Y 580.241,Z 185.518,A -85,B 0,C 180,E1 -1936.613,E2 -1936.613} C_VEL
LIN {X 0,Y 580.292,Z 185.514,A -85,B 0,C 180,E1 -1939.156,E2 -1939.156} C_VEL
LIN {X 0,Y 580.282,Z 185.51,A -85,B 0,C 180,E1 -1941.927,E2 -1941.927} C_VEL
LIN {X 0,Y 580.246,Z 185.516,A -85,B 0,C 180,E1 -1944.452,E2 -1944.452} C_VEL
LIN {X 0,Y 580.285,Z 185.515,A -85,B 0,C 180,E1 -1946.975,E2 -1946.975} C_VEL
LIN {X 0,Y 580.286,Z 185.51,A -85,B 0,C 180,E1 -1949.425,E2 -1949.425} C_VEL
LIN {X 0,Y 580.293,Z 185.51,A -85,B 0,C 180,E1 -1952.141,E2 -1952.141} C_VEL
LIN {X 0,Y 580.316,Z 185.506,A -85,B 0,C 180,E1 -1955.27,E2 -1955.27} C_VEL
LIN {X 0,Y 580.265,Z 185.513,A -85,B 0,C 180,E1 -1957.947,E2 -1957.947} C_VEL
LIN {X 0,Y 580.295,Z 185.511,A -85,B 0,C 180,E1 -1960.913,E2 -1960.913} C_VEL
LIN {X 0,Y 580.268,Z 185.512,A -85,B 0,C 180,E1 -1963.825,E2 -1963.825} C_VEL
LIN {X 0,Y 580.313,Z 185.508,A -85,B 0,C 180,E1 -1965.983,E2 -1965.983} C_VEL
LIN {X 0,Y 580.301,Z 185.509,A -85,B 0,C 180,E1 -1968.827,E2 -1968.827} C_VEL
LIN {X 0,Y 580.305,Z 185.507,A -85,B 0,C 180,E1 -1971.644,E2 -1971.644} C_VEL
LIN {X 0,Y 580.319,Z 185.512,A -85,B 0,C 180,E1 -1974.44,E2 -1974.44} C_VEL
LIN {X 0,Y 580.332,Z 185.499,A -85,B 0,C 180,E1 -1977.223,E2 -1977.223} C_VEL
LIN {X 0,Y 580.344,Z 185.506,A -85,B 0,C 180,E1 -1980,E2 -1980} C_VEL
LIN {X 0,Y 580.338,Z 185.504,A -85,B 0,C 180,E1 -1982.777,E2 -1982.777} C_VEL
LIN {X 0,Y 580.314,Z 185.504,A -85,B 0,C 180,E1 -1985.56,E2 -1985.56} C_VEL
LIN {X 0,Y 580.324,Z 185.51,A -85,B 0,C 180,E1 -1988.356,E2 -1988.356} C_VEL
LIN {X 0,Y 580.296,Z 185.506,A -85,B 0,C 180,E1 -1991.191,E2 -1991.191} C_VEL
LIN {X 0,Y 580.322,Z 185.513,A -85,B 0,C 180,E1 -1994.017,E2 -1994.017} C_VEL
LIN {X 0,Y 580.309,Z 185.505,A -85,B 0,C 180,E1 -1996.914,E2 -1996.914} C_VEL
LIN {X 0,Y 580.302,Z 185.513,A -85,B 0,C 180,E1 -1999.822,E2 -1999.822} C_VEL
LIN {X 0,Y 580.279,Z 185.511,A -85,B 0,C 180,E1 -2001.336,E2 -2001.336} C_VEL
LIN {X 0,Y 579.583,Z 185.607,A -85,B 0,C 180,E1 -2001.915,E2 -2001.915} C_VEL
LIN {X 0,Y 576.707,Z 185.96,A -85,B 0,C 180,E1 -2002.855,E2 -2002.855} C_VEL
LIN {X 0,Y 574.313,Z 186.258,A -85,B 0,C 180,E1 -2003.611,E2 -2003.611} C_VEL
LIN {X 0,Y 573.314,Z 186.381,A -85,B 0,C 180,E1 -2004.195,E2 -2004.195} C_VEL
LIN {X 0,Y 573.248,Z 186.386,A -85,B 0,C 180,E1 -2004.392,E2 -2004.392} C_VEL
LIN {X 0,Y 573.247,Z 186.385,A -85,B 0,C 180,E1 -2006.976,E2 -2006.976} C_VEL
LIN {X 0,Y 573.25,Z 186.391,A -85,B 0,C 180,E1 -2009.489,E2 -2009.489} C_VEL
LIN {X 0,Y 573.252,Z 186.383,A -85,B 0,C 180,E1 -2012.645,E2 -2012.645} C_VEL
LIN {X 0,Y 573.265,Z 186.386,A -85,B 0,C 180,E1 -2015.184,E2 -2015.184} C_VEL
LIN {X 0,Y 573.233,Z 186.393,A -85,B 0,C 180,E1 -2017.808,E2 -2017.808} C_VEL
LIN {X 0,Y 573.241,Z 186.387,A -85,B 0,C 180,E1 -2020.525,E2 -2020.525} C_VEL
LIN {X 0,Y 573.234,Z 186.394,A -85,B 0,C 180,E1 -2023.359,E2 -2023.359} C_VEL
LIN {X 0,Y 573.242,Z 186.387,A -85,B 0,C 180,E1 -2026.331,E2 -2026.331} C_VEL
LIN {X 0,Y 573.232,Z 186.386,A -85,B 0,C 180,E1 -2028.544,E2 -2028.544} C_VEL
LIN {X 0,Y 573.24,Z 186.395,A -85,B 0,C 180,E1 -2031.299,E2 -2031.299} C_VEL
LIN {X 0,Y 573.213,Z 186.39,A -85,B 0,C 180,E1 -2034.018,E2 -2034.018} C_VEL
LIN {X 0,Y 573.284,Z 186.382,A -85,B 0,C 180,E1 -2036.519,E2 -2036.519} C_VEL
LIN {X 0,Y 573.232,Z 186.394,A -85,B 0,C 180,E1 -2039.117,E2 -2039.117} C_VEL
LIN {X 0,Y 573.25,Z 186.385,A -85,B 0,C 180,E1 -2041.971,E2 -2041.971} C_VEL
LIN {X 0,Y 573.256,Z 186.387,A -85,B 0,C 180,E1 -2044.59,E2 -2044.59} C_VEL
LIN {X 0,Y 573.235,Z 186.39,A -85,B 0,C 180,E1 -2047.662,E2 -2047.662} C_VEL
LIN {X 0,Y 573.265,Z 186.385,A -85,B 0,C 180,E1 -2050.67,E2 -2050.67} C_VEL
LIN {X 0,Y 573.241,Z 186.389,A -85,B 0,C 180,E1 -2053.621,E2 -2053.621} C_VEL
LIN {X 0,Y 573.273,Z 186.38,A -85,B 0,C 180,E1 -2055.807,E2 -2055.807} C_VEL
LIN {X 0,Y 573.263,Z 186.391,A -85,B 0,C 180,E1 -2058.745,E2 -2058.745} C_VEL
LIN {X 0,Y 573.282,Z 186.384,A -85,B 0,C 180,E1 -2061.54,E2 -2061.54} C_VEL
LIN {X 0,Y 573.297,Z 186.382,A -85,B 0,C 180,E1 -2064.372,E2 -2064.372} C_VEL
LIN {X 0,Y 573.313,Z 186.38,A -85,B 0,C 180,E1 -2067.892,E2 -2067.892} C_VEL
LIN {X 0,Y 573.323,Z 186.404,A -85,B 0,C 180,E1 -2070.373,E2 -2070.373} C_VEL
LIN {X 0,Y 574.992,Z 194.088,A -85,B 0,C 180,E1 -2071.225,E2 -2071.225} C_VEL
LIN {X 0,Y 574.809,Z 205.917,A -85,B 0,C 180,E1 -2072.383,E2 -2072.383} C_VEL
LIN {X 0,Y 576.21,Z 213.409,A -85,B 0,C 180,E1 -2072.544,E2 -2072.544} C_VEL
LIN {X 0,Y 575.549,Z 411.033,A -85,B 0,C 180,E1 -2075.145,E2 -2075.145} C_VEL
LIN {X 0,Y 575.377,Z 427.664,A -85,B 0,C 180,E1 -2075.498,E2 -2075.498} C_VEL
LIN {X 0,Y 575.149,Z 443.187,A -85,B 0,C 180,E1 -2075.962,E2 -2075.962} C_VEL
LIN {X 0,Y 574.952,Z 458.963,A -85,B 0,C 180,E1 -2076.58,E2 -2076.58} C_VEL
LIN {X 0,Y 574.618,Z 475.329,A -85,B 0,C 180,E1 -2077.39,E2 -2077.39} C_VEL
LIN {X 0,Y 574.366,Z 489.488,A -85,B 0,C 180,E1 -2078.248,E2 -2078.248} C_VEL
LIN {X 0,Y 574.095,Z 503.362,A -85,B 0,C 180,E1 -2079.246,E2 -2079.246} C_VEL
LIN {X 0,Y 573.825,Z 517.012,A -85,B 0,C 180,E1 -2080.407,E2 -2080.407} C_VEL
LIN {X 0,Y 573.587,Z 529.189,A -85,B 0,C 180,E1 -2081.628,E2 -2081.628} C_VEL
LIN {X 0,Y 573.44,Z 540.227,A -85,B 0,C 180,E1 -2082.924,E2 -2082.924} C_VEL
LIN {X 0,Y 573.264,Z 550.955,A -85,B 0,C 180,E1 -2084.418,E2 -2084.418} C_VEL
LIN {X 0,Y 573.15,Z 559.449,A -85,B 0,C 180,E1 -2085.832,E2 -2085.832} C_VEL
LIN {X 0,Y 573.107,Z 565.987,A -85,B 0,C 180,E1 -2087.116,E2 -2087.116} C_VEL
LIN {X 0,Y 573.052,Z 572.258,A -85,B 0,C 180,E1 -2088.594,E2 -2088.594} C_VEL
LIN {X 0,Y 573.008,Z 577.261,A -85,B 0,C 180,E1 -2090.085,E2 -2090.085} C_VEL
LIN {X 0,Y 572.938,Z 581.159,A -85,B 0,C 180,E1 -2091.592,E2 -2091.592} C_VEL
LIN {X 0,Y 572.93,Z 583.899,A -85,B 0,C 180,E1 -2093.112,E2 -2093.112} C_VEL
LIN {X 0,Y 572.9,Z 585.585,A -85,B 0,C 180,E1 -2094.799,E2 -2094.799} C_VEL
LIN {X 0,Y 572.951,Z 585.92,A -85,B 0,C 180,E1 -2096.435,E2 -2096.435} C_VEL
LIN {X 0,Y 572.934,Z 585.097,A -85,B 0,C 180,E1 -2097.97,E2 -2097.97} C_VEL
LIN {X 0,Y 572.967,Z 583.175,A -85,B 0,C 180,E1 -2099.439,E2 -2099.439} C_VEL
LIN {X 0,Y 572.982,Z 579.964,A -85,B 0,C 180,E1 -2101.007,E2 -2101.007} C_VEL
LIN {X 0,Y 572.978,Z 575.215,A -85,B 0,C 180,E1 -2102.662,E2 -2102.662} C_VEL
LIN {X 0,Y 573.043,Z 570.571,A -85,B 0,C 180,E1 -2103.919,E2 -2103.919} C_VEL
LIN {X 0,Y 573.097,Z 564.968,A -85,B 0,C 180,E1 -2105.195,E2 -2105.195} C_VEL
LIN {X 0,Y 573.141,Z 556.894,A -85,B 0,C 180,E1 -2106.711,E2 -2106.711} C_VEL
LIN {X 0,Y 573.305,Z 548.312,A -85,B 0,C 180,E1 -2108.061,E2 -2108.061} C_VEL
LIN {X 0,Y 573.455,Z 537.86,A -85,B 0,C 180,E1 -2109.458,E2 -2109.458} C_VEL
LIN {X 0,Y 573.633,Z 526.703,A -85,B 0,C 180,E1 -2110.728,E2 -2110.728} C_VEL
LIN {X 0,Y 573.878,Z 514.026,A -85,B 0,C 180,E1 -2111.958,E2 -2111.958} C_VEL
LIN {X 0,Y 574.177,Z 499.931,A -85,B 0,C 180,E1 -2113.112,E2 -2113.112} C_VEL
LIN {X 0,Y 574.444,Z 485.79,A -85,B 0,C 180,E1 -2114.082,E2 -2114.082} C_VEL
LIN {X 0,Y 574.744,Z 471.115,A -85,B 0,C 180,E1 -2114.922,E2 -2114.922} C_VEL
LIN {X 0,Y 574.977,Z 456.334,A -85,B 0,C 180,E1 -2115.621,E2 -2115.621} C_VEL
LIN {X 0,Y 575.217,Z 440.07,A -85,B 0,C 180,E1 -2116.232,E2 -2116.232} C_VEL
LIN {X 0,Y 575.418,Z 423.271,A -85,B 0,C 180,E1 -2116.704,E2 -2116.704} C_VEL
LIN {X 0,Y 575.547,Z 405.979,A -85,B 0,C 180,E1 -2117.028,E2 -2117.028} C_VEL
LIN {X 0,Y 576.166,Z 213.033,A -85,B 0,C 180,E1 -2119.553,E2 -2119.553} C_VEL
LIN {X 0,Y 574.768,Z 205.851,A -85,B 0,C 180,E1 -2119.713,E2 -2119.713} C_VEL
LIN {X 0,Y 574.868,Z 192.994,A -85,B 0,C 180,E1 -2120.979,E2 -2120.979} C_VEL
LIN {X 0,Y 573.222,Z 186.397,A -85,B 0,C 180,E1 -2121.751,E2 -2121.751} C_VEL
LIN {X 0,Y 573.184,Z 186.397,A -85,B 0,C 180,E1 -2124.021,E2 -2124.021} C_VEL
LIN {X 0,Y 573.219,Z 186.391,A -85,B 0,C 180,E1 -2126.515,E2 -2126.515} C_VEL
LIN {X 0,Y 573.211,Z 186.4,A -85,B 0,C 180,E1 -2129.119,E2 -2129.119} C_VEL
LIN {X 0,Y 573.214,Z 186.391,A -85,B 0,C 180,E1 -2131.976,E2 -2131.976} C_VEL
LIN {X 0,Y 573.217,Z 186.394,A -85,B 0,C 180,E1 -2134.588,E2 -2134.588} C_VEL
LIN {X 0,Y 573.216,Z 186.39,A -85,B 0,C 180,E1 -2137.661,E2 -2137.661} C_VEL
LIN {X 0,Y 573.23,Z 186.389,A -85,B 0,C 180,E1 -2139.923,E2 -2139.923} C_VEL
LIN {X 0,Y 573.252,Z 186.391,A -85,B 0,C 180,E1 -2142.99,E2 -2142.99} C_VEL
LIN {X 0,Y 573.257,Z 186.385,A -85,B 0,C 180,E1 -2145.807,E2 -2145.807} C_VEL
LIN {X 0,Y 573.255,Z 186.393,A -85,B 0,C 180,E1 -2148.745,E2 -2148.745} C_VEL
LIN {X 0,Y 573.245,Z 186.386,A -85,B 0,C 180,E1 -2151.54,E2 -2151.54} C_VEL
LIN {X 0,Y 573.228,Z 186.388,A -85,B 0,C 180,E1 -2153.665,E2 -2153.665} C_VEL
LIN {X 0,Y 573.21,Z 186.392,A -85,B 0,C 180,E1 -2155.781,E2 -2155.781} C_VEL
LIN {X 0,Y 573.295,Z 186.383,A -85,B 0,C 180,E1 -2157.892,E2 -2157.892} C_VEL
LIN {X 0,Y 573.331,Z 186.379,A -85,B 0,C 180,E1 -2160.702,E2 -2160.702} C_VEL
LIN {X 0,Y 573.226,Z 186.389,A -85,B 0,C 180,E1 -2163.515,E2 -2163.515} C_VEL
LIN {X 0,Y 573.28,Z 186.384,A -85,B 0,C 180,E1 -2165.628,E2 -2165.628} C_VEL
LIN {X 0,Y 573.283,Z 186.386,A -85,B 0,C 180,E1 -2168.459,E2 -2168.459} C_VEL
LIN {X 0,Y 573.264,Z 186.384,A -85,B 0,C 180,E1 -2171.312,E2 -2171.312} C_VEL
LIN {X 0,Y 573.267,Z 186.39,A -85,B 0,C 180,E1 -2174.193,E2 -2174.193} C_VEL
LIN {X 0,Y 573.253,Z 186.386,A -85,B 0,C 180,E1 -2177.112,E2 -2177.112} C_VEL
LIN {X 0,Y 573.246,Z 186.392,A -85,B 0,C 180,E1 -2180.077,E2 -2180.077} C_VEL
LIN {X 0,Y 573.227,Z 186.39,A -85,B 0,C 180,E1 -2183.1,E2 -2183.1} C_VEL
LIN {X 0,Y 573.251,Z 186.391,A -85,B 0,C 180,E1 -2185.41,E2 -2185.41} C_VEL
LIN {X 0,Y 573.258,Z 186.388,A -85,B 0,C 180,E1 -2188.032,E2 -2188.032} C_VEL
LIN {X 0,Y 573.232,Z 186.39,A -85,B 0,C 180,E1 -2190.884,E2 -2190.884} C_VEL
LIN {X 0,Y 573.283,Z 186.391,A -85,B 0,C 180,E1 -2193.528,E2 -2193.528} C_VEL
LIN {X 0,Y 573.209,Z 186.393,A -85,B 0,C 180,E1 -2196.052,E2 -2196.052} C_VEL
LIN {X 0,Y 573.241,Z 186.389,A -85,B 0,C 180,E1 -2198.701,E2 -2198.701} C_VEL
LIN {X 0,Y 573.225,Z 186.396,A -85,B 0,C 180,E1 -2201.457,E2 -2201.457} C_VEL
LIN {X 0,Y 573.23,Z 186.39,A -85,B 0,C 180,E1 -2204.334,E2 -2204.334} C_VEL
LIN {X 0,Y 573.235,Z 186.394,A -85,B 0,C 180,E1 -2207.359,E2 -2207.359} C_VEL
LIN {X 0,Y 573.245,Z 186.39,A -85,B 0,C 180,E1 -2210.568,E2 -2210.568} C_VEL
LIN {X 0,Y 573.247,Z 186.395,A -85,B 0,C 180,E1 -2213.078,E2 -2213.078} C_VEL
LIN {X 0,Y 573.26,Z 186.385,A -85,B 0,C 180,E1 -2215.672,E2 -2215.672} C_VEL
LIN {X 0,Y 573.239,Z 186.39,A -85,B 0,C 180,E1 -2218.185,E2 -2218.185} C_VEL
LIN {X 0,Y 573.25,Z 186.395,A -85,B 0,C 180,E1 -2220.634,E2 -2220.634} C_VEL
LIN {X 0,Y 573.291,Z 186.589,A -85,B 0,C 180,E1 -2222.005,E2 -2222.005} C_VEL
LIN {X 0,Y 575.475,Z 194.158,A -85,B 0,C 180,E1 -2222.784,E2 -2222.784} C_VEL
LIN {X 0,Y 575.305,Z 215.971,A -85,B 0,C 180,E1 -2224.688,E2 -2224.688} C_VEL
LIN {X 0,Y 575.032,Z 234.96,A -85,B 0,C 180,E1 -2226.329,E2 -2226.329} C_VEL
LIN {X 0,Y 576.214,Z 242.189,A -85,B 0,C 180,E1 -2226.483,E2 -2226.483} C_VEL
LIN {X 0,Y 575.5,Z 442.456,A -85,B 0,C 180,E1 -2229.119,E2 -2229.119} C_VEL
LIN {X 0,Y 575.356,Z 459.025,A -85,B 0,C 180,E1 -2229.488,E2 -2229.488} C_VEL
LIN {X 0,Y 575.126,Z 475.255,A -85,B 0,C 180,E1 -2229.992,E2 -2229.992} C_VEL
LIN {X 0,Y 574.881,Z 491.205,A -85,B 0,C 180,E1 -2230.639,E2 -2230.639} C_VEL
LIN {X 0,Y 574.661,Z 505.725,A -85,B 0,C 180,E1 -2231.368,E2 -2231.368} C_VEL
LIN {X 0,Y 574.367,Z 520.658,A -85,B 0,C 180,E1 -2232.278,E2 -2232.278} C_VEL
LIN {X 0,Y 574.103,Z 534.389,A -85,B 0,C 180,E1 -2233.281,E2 -2233.281} C_VEL
LIN {X 0,Y 573.83,Z 547.075,A -85,B 0,C 180,E1 -2234.369,E2 -2234.369} C_VEL
LIN {X 0,Y 573.603,Z 559.283,A -85,B 0,C 180,E1 -2235.595,E2 -2235.595} C_VEL
LIN {X 0,Y 573.418,Z 570.339,A -85,B 0,C 180,E1 -2236.895,E2 -2236.895} C_VEL
LIN {X 0,Y 573.282,Z 580.675,A -85,B 0,C 180,E1 -2238.33,E2 -2238.33} C_VEL
LIN {X 0,Y 573.168,Z 589.286,A -85,B 0,C 180,E1 -2239.759,E2 -2239.759} C_VEL
LIN {X 0,Y 573.076,Z 596.49,A -85,B 0,C 180,E1 -2241.182,E2 -2241.182} C_VEL
LIN {X 0,Y 573.039,Z 602.468,A -85,B 0,C 180,E1 -2242.601,E2 -2242.601} C_VEL
LIN {X 0,Y 573.016,Z 607.187,A -85,B 0,C 180,E1 -2244.016,E2 -2244.016} C_VEL
LIN {X 0,Y 573.005,Z 611.637,A -85,B 0,C 180,E1 -2245.78,E2 -2245.78} C_VEL
LIN {X 0,Y 572.947,Z 614.089,A -85,B 0,C 180,E1 -2247.188,E2 -2247.188} C_VEL
LIN {X 0,Y 572.939,Z 615.48,A -85,B 0,C 180,E1 -2248.594,E2 -2248.594} C_VEL
LIN {X 0,Y 572.933,Z 616,A -85,B 0,C 180,E1 -2250,E2 -2250} C_VEL
LIN {X 0,Y 572.939,Z 615.479,A -85,B 0,C 180,E1 -2251.406,E2 -2251.406} C_VEL
LIN {X 0,Y 572.947,Z 614.088,A -85,B 0,C 180,E1 -2252.813,E2 -2252.813} C_VEL
LIN {X 0,Y 573.006,Z 611.635,A -85,B 0,C 180,E1 -2254.22,E2 -2254.22} C_VEL
LIN {X 0,Y 573.015,Z 607.187,A -85,B 0,C 180,E1 -2255.984,E2 -2255.984} C_VEL
LIN {X 0,Y 573.04,Z 602.468,A -85,B 0,C 180,E1 -2257.399,E2 -2257.399} C_VEL
LIN {X 0,Y 573.077,Z 596.488,A -85,B 0,C 180,E1 -2258.818,E2 -2258.818} C_VEL
LIN {X 0,Y 573.181,Z 588.276,A -85,B 0,C 180,E1 -2260.42,E2 -2260.42} C_VEL
LIN {X 0,Y 573.269,Z 579.443,A -85,B 0,C 180,E1 -2261.85,E2 -2261.85} C_VEL
